LIN {X 0,Y 523.96,Z 519.214,A -85,B 0,C 180,E1 -4880.41,E2 -4880.41} C_VEL
LIN {X 0,Y 523.905,Z 519.224,A -85,B 0,C 180,E1 -4882.893,E2 -4882.893} C_VEL
LIN {X 0,Y 523.943,Z 519.224,A -85,B 0,C 180,E1 -4885.419,E2 -4885.419} C_VEL
LIN {X 0,Y 523.959,Z 519.22,A -85,B 0,C 180,E1 -4887.999,E2 -4887.999} C_VEL
LIN {X 0,Y 523.998,Z 519.419,A -85,B 0,C 180,E1 -4889.406,E2 -4889.406} C_VEL
LIN {X 0,Y 524.764,Z 524.163,A -85,B 0,C 180,E1 -4890.369,E2 -4890.369} C_VEL
LIN {X 0,Y 524.382,Z 539.428,A -85,B 0,C 180,E1 -4893.332,E2 -4893.332} C_VEL
LIN {X 0,Y 524.173,Z 547.59,A -85,B 0,C 180,E1 -4894.895,E2 -4894.895} C_VEL
LIN {X 0,Y 525.927,Z 557.88,A -85,B 0,C 180,E1 -4895.101,E2 -4895.101} C_VEL
LIN {X 0,Y 525.587,Z 637.04,A -85,B 0,C 180,E1 -4896.188,E2 -4896.188} C_VEL
LIN {X 0,Y 524.906,Z 640.968,A -85,B 0,C 180,E1 -4896.222,E2 -4896.222} C_VEL
LIN {X 0,Y 519.182,Z 653.237,A -85,B 0,C 180,E1 -4896.254,E2 -4896.254} C_VEL
LIN {X 0,Y 518.575,Z 657.117,A -85,B 0,C 180,E1 -4896.319,E2 -4896.319} C_VEL
LIN {X 0,Y 518.341,Z 670.235,A -85,B 0,C 180,E1 -4896.688,E2 -4896.688} C_VEL
LIN {X 0,Y 518.086,Z 682.787,A -85,B 0,C 180,E1 -4897.211,E2 -4897.211} C_VEL
LIN {X 0,Y 517.827,Z 694.371,A -85,B 0,C 180,E1 -4897.855,E2 -4897.855} C_VEL
LIN {X 0,Y 517.513,Z 705.687,A -85,B 0,C 180,E1 -4898.659,E2 -4898.659} C_VEL
LIN {X 0,Y 517.226,Z 715.845,A -85,B 0,C 180,E1 -4899.565,E2 -4899.565} C_VEL
LIN {X 0,Y 516.953,Z 724.842,A -85,B 0,C 180,E1 -4900.548,E2 -4900.548} C_VEL
LIN {X 0,Y 516.741,Z 732.6,A -85,B 0,C 180,E1 -4901.582,E2 -4901.582} C_VEL
LIN {X 0,Y 516.508,Z 740.372,A -85,B 0,C 180,E1 -4902.869,E2 -4902.869} C_VEL
LIN {X 0,Y 516.368,Z 746.561,A -85,B 0,C 180,E1 -4904.175,E2 -4904.175} C_VEL
LIN {X 0,Y 516.289,Z 751.444,A -85,B 0,C 180,E1 -4905.541,E2 -4905.541} C_VEL
LIN {X 0,Y 516.239,Z 754.36,A -85,B 0,C 180,E1 -4906.641,E2 -4906.641} C_VEL
LIN {X 0,Y 516.182,Z 756.998,A -85,B 0,C 180,E1 -4908.154,E2 -4908.154} C_VEL
LIN {X 0,Y 516.14,Z 758.095,A -85,B 0,C 180,E1 -4909.686,E2 -4909.686} C_VEL
LIN {X 0,Y 516.129,Z 757.71,A -85,B 0,C 180,E1 -4911.219,E2 -4911.219} C_VEL
LIN {X 0,Y 516.154,Z 756.609,A -85,B 0,C 180,E1 -4912.215,E2 -4912.215} C_VEL
LIN {X 0,Y 516.236,Z 754.376,A -85,B 0,C 180,E1 -4913.438,E2 -4913.438} C_VEL
LIN {X 0,Y 516.246,Z 750.774,A -85,B 0,C 180,E1 -4914.767,E2 -4914.767} C_VEL
LIN {X 0,Y 516.383,Z 745.673,A -85,B 0,C 180,E1 -4916.12,E2 -4916.12} C_VEL
LIN {X 0,Y 516.563,Z 738.759,A -85,B 0,C 180,E1 -4917.514,E2 -4917.514} C_VEL
LIN {X 0,Y 516.756,Z 731.562,A -85,B 0,C 180,E1 -4918.655,E2 -4918.655} C_VEL
LIN {X 0,Y 516.994,Z 722.592,A -85,B 0,C 180,E1 -4919.804,E2 -4919.804} C_VEL
LIN {X 0,Y 517.265,Z 712.654,A -85,B 0,C 180,E1 -4920.83,E2 -4920.83} C_VEL
LIN {X 0,Y 517.605,Z 701.844,A -85,B 0,C 180,E1 -4921.723,E2 -4921.723} C_VEL
LIN {X 0,Y 517.9,Z 691.117,A -85,B 0,C 180,E1 -4922.434,E2 -4922.434} C_VEL
LIN {X 0,Y 518.189,Z 679.448,A -85,B 0,C 180,E1 -4923.033,E2 -4923.033} C_VEL
LIN {X 0,Y 518.403,Z 666.182,A -85,B 0,C 180,E1 -4923.534,E2 -4923.534} C_VEL
LIN {X 0,Y 518.597,Z 653.698,A -85,B 0,C 180,E1 -4923.843,E2 -4923.843} C_VEL
LIN {X 0,Y 519.061,Z 558.357,A -85,B 0,C 180,E1 -4925.184,E2 -4925.184} C_VEL
LIN {X 0,Y 517.217,Z 547.636,A -85,B 0,C 180,E1 -4925.419,E2 -4925.419} C_VEL
LIN {X 0,Y 517.535,Z 532.885,A -85,B 0,C 180,E1 -4928.283,E2 -4928.283} C_VEL
LIN {X 0,Y 517.722,Z 524.988,A -85,B 0,C 180,E1 -4929.828,E2 -4929.828} C_VEL
LIN {X 0,Y 516.919,Z 520.098,A -85,B 0,C 180,E1 -4930.854,E2 -4930.854} C_VEL
LIN {X 0,Y 516.911,Z 520.095,A -85,B 0,C 180,E1 -4933.411,E2 -4933.411} C_VEL
LIN {X 0,Y 516.891,Z 520.095,A -85,B 0,C 180,E1 -4935.835,E2 -4935.835} C_VEL
LIN {X 0,Y 516.96,Z 520.086,A -85,B 0,C 180,E1 -4938.235,E2 -4938.235} C_VEL
LIN {X 0,Y 516.965,Z 520.086,A -85,B 0,C 180,E1 -4941.401,E2 -4941.401} C_VEL
LIN {X 0,Y 516.999,Z 520.08,A -85,B 0,C 180,E1 -4943.758,E2 -4943.758} C_VEL
LIN {X 0,Y 517.012,Z 520.088,A -85,B 0,C 180,E1 -4946.884,E2 -4946.884} C_VEL
LIN {X 0,Y 517.083,Z 520.069,A -85,B 0,C 180,E1 -4950.001,E2 -4950.001} C_VEL
LIN {X 0,Y 517.011,Z 520.085,A -85,B 0,C 180,E1 -4953.118,E2 -4953.118} C_VEL
LIN {X 0,Y 517,Z 520.08,A -85,B 0,C 180,E1 -4956.244,E2 -4956.244} C_VEL
LIN {X 0,Y 516.95,Z 520.09,A -85,B 0,C 180,E1 -4959.39,E2 -4959.39} C_VEL
LIN {X 0,Y 516.951,Z 520.086,A -85,B 0,C 180,E1 -4961.809,E2 -4961.809} C_VEL
LIN {X 0,Y 516.944,Z 520.095,A -85,B 0,C 180,E1 -4965.148,E2 -4965.148} C_VEL
LIN {X 0,Y 516.916,Z 520.09,A -85,B 0,C 180,E1 -4968.224,E2 -4968.224} C_VEL
LIN {X 0,Y 516.913,Z 520.094,A -85,B 0,C 180,E1 -4970.702,E2 -4970.702} C_VEL
LIN {X 0,Y 516.891,Z 520.093,A -85,B 0,C 180,E1 -4974.074,E2 -4974.074} C_VEL
LIN {X 0,Y 516.925,Z 520.091,A -85,B 0,C 180,E1 -4976.659,E2 -4976.659} C_VEL
LIN {X 0,Y 516.912,Z 520.095,A -85,B 0,C 180,E1 -4979.525,E2 -4979.525} C_VEL
LIN {X 0,Y 516.897,Z 520.093,A -85,B 0,C 180,E1 -4982.544,E2 -4982.544} C_VEL
LIN {X 0,Y 516.867,Z 520.105,A -85,B 0,C 180,E1 -4985.331,E2 -4985.331} C_VEL
LIN {X 0,Y 516.883,Z 520.095,A -85,B 0,C 180,E1 -4987.944,E2 -4987.944} C_VEL
LIN {X 0,Y 516.888,Z 520.095,A -85,B 0,C 180,E1 -4990.742,E2 -4990.742} C_VEL
LIN {X 0,Y 516.908,Z 520.093,A -85,B 0,C 180,E1 -4992.83,E2 -4992.83} C_VEL
LIN {X 0,Y 516.925,Z 520.093,A -85,B 0,C 180,E1 -4995.011,E2 -4995.011} C_VEL
LIN {X 0,Y 516.918,Z 520.09,A -85,B 0,C 180,E1 -4998.399,E2 -4998.399} C_VEL
LIN {X 0,Y 516.885,Z 520.101,A -85,B 0,C 180,E1 -5001.285,E2 -5001.285} C_VEL
LIN {X 0,Y 516.875,Z 520.096,A -85,B 0,C 180,E1 -5004.221,E2 -5004.221} C_VEL
LIN {X 0,Y 516.9,Z 520.095,A -85,B 0,C 180,E1 -5007.054,E2 -5007.054} C_VEL
LIN {X 0,Y 516.896,Z 520.098,A -85,B 0,C 180,E1 -5009.797,E2 -5009.797} C_VEL
LIN {X 0,Y 516.93,Z 520.088,A -85,B 0,C 180,E1 -5012.468,E2 -5012.468} C_VEL
LIN {X 0,Y 516.913,Z 520.093,A -85,B 0,C 180,E1 -5015.073,E2 -5015.073} C_VEL
LIN {X 0,Y 516.89,Z 520.093,A -85,B 0,C 180,E1 -5018.463,E2 -5018.463} C_VEL
LIN {X 0,Y 516.905,Z 520.092,A -85,B 0,C 180,E1 -5020.955,E2 -5020.955} C_VEL
LIN {X 0,Y 516.914,Z 520.096,A -85,B 0,C 180,E1 -5023.411,E2 -5023.411} C_VEL
LIN {X 0,Y 516.901,Z 520.099,A -85,B 0,C 180,E1 -5025.834,E2 -5025.834} C_VEL
LIN {X 0,Y 516.972,Z 520.085,A -85,B 0,C 180,E1 -5028.234,E2 -5028.234} C_VEL
LIN {X 0,Y 516.971,Z 520.087,A -85,B 0,C 180,E1 -5031.4,E2 -5031.4} C_VEL
LIN {X 0,Y 517.016,Z 520.087,A -85,B 0,C 180,E1 -5033.757,E2 -5033.757} C_VEL
LIN {X 0,Y 517.089,Z 520.076,A -85,B 0,C 180,E1 -5037.664,E2 -5037.664} C_VEL
LIN {X 0,Y 517.1,Z 520.067,A -85,B 0,C 180,E1 -5040.779,E2 -5040.779} C_VEL
LIN {X 0,Y 517.018,Z 520.078,A -85,B 0,C 180,E1 -5043.117,E2 -5043.117} C_VEL
LIN {X 0,Y 517.017,Z 520.082,A -85,B 0,C 180,E1 -5046.243,E2 -5046.243} C_VEL
LIN {X 0,Y 516.951,Z 520.088,A -85,B 0,C 180,E1 -5049.39,E2 -5049.39} C_VEL
LIN {X 0,Y 516.96,Z 520.092,A -85,B 0,C 180,E1 -5051.807,E2 -5051.807} C_VEL
LIN {X 0,Y 516.952,Z 520.086,A -85,B 0,C 180,E1 -5055.147,E2 -5055.147} C_VEL
LIN {X 0,Y 516.924,Z 520.095,A -85,B 0,C 180,E1 -5058.223,E2 -5058.223} C_VEL
LIN {X 0,Y 516.92,Z 520.091,A -85,B 0,C 180,E1 -5060.702,E2 -5060.702} C_VEL
LIN {X 0,Y 516.898,Z 520.102,A -85,B 0,C 180,E1 -5064.073,E2 -5064.073} C_VEL
LIN {X 0,Y 516.93,Z 520.09,A -85,B 0,C 180,E1 -5066.658,E2 -5066.658} C_VEL
LIN {X 0,Y 516.919,Z 520.091,A -85,B 0,C 180,E1 -5069.524,E2 -5069.524} C_VEL
LIN {X 0,Y 516.901,Z 520.096,A -85,B 0,C 180,E1 -5072.543,E2 -5072.543} C_VEL
LIN {X 0,Y 516.884,Z 520.094,A -85,B 0,C 180,E1 -5075.331,E2 -5075.331} C_VEL
LIN {X 0,Y 516.888,Z 520.099,A -85,B 0,C 180,E1 -5077.943,E2 -5077.943} C_VEL
LIN {X 0,Y 516.889,Z 520.096,A -85,B 0,C 180,E1 -5080.742,E2 -5080.742} C_VEL
LIN {X 0,Y 516.888,Z 520.097,A -85,B 0,C 180,E1 -5083.903,E2 -5083.903} C_VEL
LIN {X 0,Y 516.889,Z 520.1,A -85,B 0,C 180,E1 -5086.107,E2 -5086.107} C_VEL
LIN {X 0,Y 516.921,Z 520.098,A -85,B 0,C 180,E1 -5088.398,E2 -5088.398} C_VEL
LIN {X 0,Y 516.887,Z 520.094,A -85,B 0,C 180,E1 -5091.284,E2 -5091.284} C_VEL
LIN {X 0,Y 516.878,Z 520.102,A -85,B 0,C 180,E1 -5094.219,E2 -5094.219} C_VEL
LIN {X 0,Y 516.902,Z 520.093,A -85,B 0,C 180,E1 -5097.052,E2 -5097.052} C_VEL
LIN {X 0,Y 516.899,Z 520.095,A -85,B 0,C 180,E1 -5099.796,E2 -5099.796} C_VEL
LIN {X 0,Y 516.934,Z 520.096,A -85,B 0,C 180,E1 -5102.467,E2 -5102.467} C_VEL
LIN {X 0,Y 516.925,Z 520.096,A -85,B 0,C 180,E1 -5105.397,E2 -5105.397} C_VEL
LIN {X 0,Y 516.918,Z 520.182,A -85,B 0,C 180,E1 -5105.595,E2 -5105.595} C_VEL
LIN {X 0,Y 518.517,Z 529.143,A -85,B 0,C 180,E1 -5107.173,E2 -5107.173} C_VEL
LIN {X 0,Y 518.016,Z 547.542,A -85,B 0,C 180,E1 -5110.172,E2 -5110.172} C_VEL
LIN {X 0,Y 517.581,Z 564.071,A -85,B 0,C 180,E1 -5112.821,E2 -5112.821} C_VEL
LIN {X 0,Y 517.335,Z 575.468,A -85,B 0,C 180,E1 -5114.64,E2 -5114.64} C_VEL
LIN {X 0,Y 519.112,Z 587.664,A -85,B 0,C 180,E1 -5114.867,E2 -5114.867} C_VEL
LIN {X 0,Y 518.603,Z 684.232,A -85,B 0,C 180,E1 -5116.23,E2 -5116.23} C_VEL
LIN {X 0,Y 518.342,Z 698.045,A -85,B 0,C 180,E1 -5116.598,E2 -5116.598} C_VEL
LIN {X 0,Y 518.105,Z 710.943,A -85,B 0,C 180,E1 -5117.115,E2 -5117.115} C_VEL
LIN {X 0,Y 517.775,Z 722.904,A -85,B 0,C 180,E1 -5117.767,E2 -5117.767} C_VEL
LIN {X 0,Y 517.531,Z 734.057,A -85,B 0,C 180,E1 -5118.544,E2 -5118.544} C_VEL
LIN {X 0,Y 517.18,Z 744.285,A -85,B 0,C 180,E1 -5119.428,E2 -5119.428} C_VEL
LIN {X 0,Y 516.953,Z 753.482,A -85,B 0,C 180,E1 -5120.412,E2 -5120.412} C_VEL
LIN {X 0,Y 516.686,Z 762.438,A -85,B 0,C 180,E1 -5121.591,E2 -5121.591} C_VEL
LIN {X 0,Y 516.512,Z 769.646,A -85,B 0,C 180,E1 -5122.768,E2 -5122.768} C_VEL
LIN {X 0,Y 516.455,Z 776.211,A -85,B 0,C 180,E1 -5124.141,E2 -5124.141} C_VEL
LIN {X 0,Y 516.272,Z 780.548,A -85,B 0,C 180,E1 -5125.314,E2 -5125.314} C_VEL
LIN {X 0,Y 516.355,Z 782.848,A -85,B 0,C 180,E1 -5126.097,E2 -5126.097} C_VEL
LIN {X 0,Y 516.283,Z 784.709,A -85,B 0,C 180,E1 -5126.878,E2 -5126.878} C_VEL
LIN {X 0,Y 516.261,Z 786.105,A -85,B 0,C 180,E1 -5127.658,E2 -5127.658} C_VEL
LIN {X 0,Y 516.16,Z 787.707,A -85,B 0,C 180,E1 -5129.219,E2 -5129.219} C_VEL
LIN {X 0,Y 516.154,Z 787.924,A -85,B 0,C 180,E1 -5129.999,E2 -5129.999} C_VEL
LIN {X 0,Y 516.192,Z 787.103,A -85,B 0,C 180,E1 -5131.559,E2 -5131.559} C_VEL
LIN {X 0,Y 516.26,Z 786.11,A -85,B 0,C 180,E1 -5132.339,E2 -5132.339} C_VEL
LIN {X 0,Y 516.282,Z 784.715,A -85,B 0,C 180,E1 -5133.12,E2 -5133.12} C_VEL
LIN {X 0,Y 516.326,Z 781.78,A -85,B 0,C 180,E1 -5134.292,E2 -5134.292} C_VEL
LIN {X 0,Y 516.405,Z 777.806,A -85,B 0,C 180,E1 -5135.465,E2 -5135.465} C_VEL
LIN {X 0,Y 516.462,Z 772.519,A -85,B 0,C 180,E1 -5136.676,E2 -5136.676} C_VEL
LIN {X 0,Y 516.596,Z 766.242,A -85,B 0,C 180,E1 -5137.818,E2 -5137.818} C_VEL
LIN {X 0,Y 516.809,Z 758.201,A -85,B 0,C 180,E1 -5138.996,E2 -5138.996} C_VEL
LIN {X 0,Y 517.023,Z 750.003,A -85,B 0,C 180,E1 -5139.979,E2 -5139.979} C_VEL
LIN {X 0,Y 517.326,Z 740.004,A -85,B 0,C 180,E1 -5140.963,E2 -5140.963} C_VEL
LIN {X 0,Y 517.655,Z 728.793,A -85,B 0,C 180,E1 -5141.842,E2 -5141.842} C_VEL
LIN {X 0,Y 517.961,Z 717.633,A -85,B 0,C 180,E1 -5142.537,E2 -5142.537} C_VEL
LIN {X 0,Y 518.237,Z 705.353,A -85,B 0,C 180,E1 -5143.128,E2 -5143.128} C_VEL
LIN {X 0,Y 518.456,Z 692.405,A -85,B 0,C 180,E1 -5143.572,E2 -5143.572} C_VEL
LIN {X 0,Y 518.687,Z 678.625,A -85,B 0,C 180,E1 -5143.865,E2 -5143.865} C_VEL
LIN {X 0,Y 518.996,Z 585.709,A -85,B 0,C 180,E1 -5145.163,E2 -5145.163} C_VEL
LIN {X 0,Y 517.345,Z 575.322,A -85,B 0,C 180,E1 -5145.367,E2 -5145.367} C_VEL
LIN {X 0,Y 517.811,Z 555.065,A -85,B 0,C 180,E1 -5148.598,E2 -5148.598} C_VEL
LIN {X 0,Y 518.244,Z 537.216,A -85,B 0,C 180,E1 -5151.477,E2 -5151.477} C_VEL
LIN {X 0,Y 518.501,Z 528.987,A -85,B 0,C 180,E1 -5152.823,E2 -5152.823} C_VEL
LIN {X 0,Y 516.92,Z 520.096,A -85,B 0,C 180,E1 -5154.406,E2 -5154.406} C_VEL
LIN {X 0,Y 516.925,Z 520.093,A -85,B 0,C 180,E1 -5156.656,E2 -5156.656} C_VEL
LIN {X 0,Y 516.909,Z 520.102,A -85,B 0,C 180,E1 -5159.523,E2 -5159.523} C_VEL
LIN {X 0,Y 516.898,Z 520.095,A -85,B 0,C 180,E1 -5162.543,E2 -5162.543} C_VEL
LIN {X 0,Y 516.876,Z 520.104,A -85,B 0,C 180,E1 -5165.331,E2 -5165.331} C_VEL
LIN {X 0,Y 516.878,Z 520.1,A -85,B 0,C 180,E1 -5167.942,E2 -5167.942} C_VEL
LIN {X 0,Y 516.881,Z 520.098,A -85,B 0,C 180,E1 -5170.74,E2 -5170.74} C_VEL
LIN {X 0,Y 516.899,Z 520.096,A -85,B 0,C 180,E1 -5172.828,E2 -5172.828} C_VEL
LIN {X 0,Y 516.916,Z 520.095,A -85,B 0,C 180,E1 -5175.009,E2 -5175.009} C_VEL
LIN {X 0,Y 516.916,Z 520.092,A -85,B 0,C 180,E1 -5178.396,E2 -5178.396} C_VEL
LIN {X 0,Y 516.88,Z 520.102,A -85,B 0,C 180,E1 -5181.284,E2 -5181.284} C_VEL
LIN {X 0,Y 516.885,Z 520.095,A -85,B 0,C 180,E1 -5184.22,E2 -5184.22} C_VEL
LIN {X 0,Y 516.89,Z 520.097,A -85,B 0,C 180,E1 -5187.052,E2 -5187.052} C_VEL
LIN {X 0,Y 516.894,Z 520.098,A -85,B 0,C 180,E1 -5189.796,E2 -5189.796} C_VEL
LIN {X 0,Y 516.921,Z 520.089,A -85,B 0,C 180,E1 -5192.467,E2 -5192.467} C_VEL
LIN {X 0,Y 516.903,Z 520.097,A -85,B 0,C 180,E1 -5195.071,E2 -5195.071} C_VEL
LIN {X 0,Y 516.877,Z 520.096,A -85,B 0,C 180,E1 -5198.461,E2 -5198.461} C_VEL
LIN {X 0,Y 516.895,Z 520.093,A -85,B 0,C 180,E1 -5200.954,E2 -5200.954} C_VEL
LIN {X 0,Y 516.908,Z 520.099,A -85,B 0,C 180,E1 -5203.41,E2 -5203.41} C_VEL
LIN {X 0,Y 516.896,Z 520.097,A -85,B 0,C 180,E1 -5205.833,E2 -5205.833} C_VEL
LIN {X 0,Y 516.993,Z 520.08,A -85,B 0,C 180,E1 -5208.234,E2 -5208.234} C_VEL
LIN {X 0,Y 516.962,Z 520.092,A -85,B 0,C 180,E1 -5211.399,E2 -5211.399} C_VEL
LIN {X 0,Y 517,Z 520.084,A -85,B 0,C 180,E1 -5213.756,E2 -5213.756} C_VEL
LIN {X 0,Y 517.007,Z 520.081,A -85,B 0,C 180,E1 -5216.883,E2 -5216.883} C_VEL
LIN {X 0,Y 517.074,Z 520.073,A -85,B 0,C 180,E1 -5220,E2 -5220} C_VEL
LIN {X 0,Y 517.007,Z 520.084,A -85,B 0,C 180,E1 -5223.117,E2 -5223.117} C_VEL
LIN {X 0,Y 516.999,Z 520.081,A -85,B 0,C 180,E1 -5226.243,E2 -5226.243} C_VEL
LIN {X 0,Y 516.947,Z 520.095,A -85,B 0,C 180,E1 -5229.389,E2 -5229.389} C_VEL
LIN {X 0,Y 516.971,Z 520.088,A -85,B 0,C 180,E1 -5231.824,E2 -5231.824} C_VEL
LIN {X 0,Y 516.931,Z 520.096,A -85,B 0,C 180,E1 -5235.146,E2 -5235.146} C_VEL
LIN {X 0,Y 516.914,Z 520.093,A -85,B 0,C 180,E1 -5238.222,E2 -5238.222} C_VEL
LIN {X 0,Y 516.901,Z 520.095,A -85,B 0,C 180,E1 -5240.701,E2 -5240.701} C_VEL
LIN {X 0,Y 516.899,Z 520.096,A -85,B 0,C 180,E1 -5244.072,E2 -5244.072} C_VEL
LIN {X 0,Y 516.917,Z 520.094,A -85,B 0,C 180,E1 -5246.658,E2 -5246.658} C_VEL
LIN {X 0,Y 516.949,Z 520.261,A -85,B 0,C 180,E1 -5249.246,E2 -5249.246} C_VEL
LIN {X 0,Y 517.804,Z 525.726,A -85,B 0,C 180,E1 -5250.37,E2 -5250.37} C_VEL
LIN {X 0,Y 517.38,Z 541.055,A -85,B 0,C 180,E1 -5253.376,E2 -5253.376} C_VEL
LIN {X 0,Y 517.2,Z 547.848,A -85,B 0,C 180,E1 -5254.694,E2 -5254.694} C_VEL
LIN {X 0,Y 519.105,Z 559.366,A -85,B 0,C 180,E1 -5254.919,E2 -5254.919} C_VEL
LIN {X 0,Y 518.611,Z 654.9,A -85,B 0,C 180,E1 -5256.271,E2 -5256.271} C_VEL
LIN {X 0,Y 518.575,Z 657.117,A -85,B 0,C 180,E1 -5256.319,E2 -5256.319} C_VEL
LIN {X 0,Y 517.98,Z 662.864,A -85,B 0,C 180,E1 -5256.446,E2 -5256.446} C_VEL
LIN {X 0,Y 515.1,Z 672.116,A -85,B 0,C 180,E1 -5256.671,E2 -5256.671} C_VEL
LIN {X 0,Y 511.993,Z 681.148,A -85,B 0,C 180,E1 -5256.969,E2 -5256.969} C_VEL
LIN {X 0,Y 511.092,Z 686.554,A -85,B 0,C 180,E1 -5257.22,E2 -5257.22} C_VEL
LIN {X 0,Y 510.843,Z 697.349,A -85,B 0,C 180,E1 -5257.874,E2 -5257.874} C_VEL
LIN {X 0,Y 510.482,Z 707.734,A -85,B 0,C 180,E1 -5258.659,E2 -5258.659} C_VEL
LIN {X 0,Y 510.18,Z 718.534,A -85,B 0,C 180,E1 -5259.678,E2 -5259.678} C_VEL
LIN {X 0,Y 509.819,Z 728.328,A -85,B 0,C 180,E1 -5260.838,E2 -5260.838} C_VEL
LIN {X 0,Y 509.594,Z 735.386,A -85,B 0,C 180,E1 -5261.866,E2 -5261.866} C_VEL
LIN {X 0,Y 509.404,Z 741.838,A -85,B 0,C 180,E1 -5263.014,E2 -5263.014} C_VEL
LIN {X 0,Y 509.296,Z 748.002,A -85,B 0,C 180,E1 -5264.411,E2 -5264.411} C_VEL
LIN {X 0,Y 509.186,Z 752.773,A -85,B 0,C 180,E1 -5265.866,E2 -5265.866} C_VEL
LIN {X 0,Y 509.095,Z 756.203,A -85,B 0,C 180,E1 -5267.436,E2 -5267.436} C_VEL
LIN {X 0,Y 509.069,Z 757.591,A -85,B 0,C 180,E1 -5268.498,E2 -5268.498} C_VEL
LIN {X 0,Y 509.057,Z 758.272,A -85,B 0,C 180,E1 -5269.545,E2 -5269.545} C_VEL
LIN {X 0,Y 509.057,Z 758.251,A -85,B 0,C 180,E1 -5270.635,E2 -5270.635} C_VEL
LIN {X 0,Y 509.064,Z 757.277,A -85,B 0,C 180,E1 -5271.898,E2 -5271.898} C_VEL
LIN {X 0,Y 509.114,Z 755.211,A -85,B 0,C 180,E1 -5273.192,E2 -5273.192} C_VEL
LIN {X 0,Y 509.183,Z 751.755,A -85,B 0,C 180,E1 -5274.572,E2 -5274.572} C_VEL
LIN {X 0,Y 509.29,Z 747.169,A -85,B 0,C 180,E1 -5275.89,E2 -5275.89} C_VEL
LIN {X 0,Y 509.455,Z 740.661,A -85,B 0,C 180,E1 -5277.298,E2 -5277.298} C_VEL
LIN {X 0,Y 509.673,Z 732.901,A -85,B 0,C 180,E1 -5278.605,E2 -5278.605} C_VEL
LIN {X 0,Y 509.945,Z 723.931,A -85,B 0,C 180,E1 -5279.801,E2 -5279.801} C_VEL
LIN {X 0,Y 510.235,Z 714.274,A -85,B 0,C 180,E1 -5280.841,E2 -5280.841} C_VEL
LIN {X 0,Y 510.563,Z 703.645,A -85,B 0,C 180,E1 -5281.759,E2 -5281.759} C_VEL
LIN {X 0,Y 510.95,Z 691.902,A -85,B 0,C 180,E1 -5282.564,E2 -5282.564} C_VEL
LIN {X 0,Y 511.282,Z 679.617,A -85,B 0,C 180,E1 -5283.208,E2 -5283.208} C_VEL
LIN {X 0,Y 511.512,Z 666.516,A -85,B 0,C 180,E1 -5283.71,E2 -5283.71} C_VEL
LIN {X 0,Y 511.725,Z 653.986,A -85,B 0,C 180,E1 -5284.026,E2 -5284.026} C_VEL
LIN {X 0,Y 512.146,Z 558.762,A -85,B 0,C 180,E1 -5285.389,E2 -5285.389} C_VEL
LIN {X 0,Y 510.224,Z 547.903,A -85,B 0,C 180,E1 -5285.621,E2 -5285.621} C_VEL
LIN {X 0,Y 510.56,Z 533.785,A -85,B 0,C 180,E1 -5288.395,E2 -5288.395} C_VEL
LIN {X 0,Y 510.76,Z 526.274,A -85,B 0,C 180,E1 -5289.881,E2 -5289.881} C_VEL
LIN {X 0,Y 509.865,Z 520.976,A -85,B 0,C 180,E1 -5290.997,E2 -5290.997} C_VEL
LIN {X 0,Y 509.879,Z 520.973,A -85,B 0,C 180,E1 -5293.176,E2 -5293.176} C_VEL
LIN {X 0,Y 509.859,Z 520.971,A -85,B 0,C 180,E1 -5295.635,E2 -5295.635} C_VEL
LIN {X 0,Y 509.897,Z 520.965,A -85,B 0,C 180,E1 -5298.124,E2 -5298.124} C_VEL
LIN {X 0,Y 509.912,Z 520.966,A -85,B 0,C 180,E1 -5301.281,E2 -5301.281} C_VEL
LIN {X 0,Y 509.95,Z 520.958,A -85,B 0,C 180,E1 -5303.671,E2 -5303.671} C_VEL
LIN {X 0,Y 509.954,Z 520.966,A -85,B 0,C 180,E1 -5306.841,E2 -5306.841} C_VEL
LIN {X 0,Y 510.061,Z 520.949,A -85,B 0,C 180,E1 -5309.212,E2 -5309.212} C_VEL
LIN {X 0,Y 510.054,Z 520.947,A -85,B 0,C 180,E1 -5312.37,E2 -5312.37} C_VEL
LIN {X 0,Y 509.977,Z 520.956,A -85,B 0,C 180,E1 -5315.537,E2 -5315.537} C_VEL
LIN {X 0,Y 509.95,Z 520.958,A -85,B 0,C 180,E1 -5317.923,E2 -5317.923} C_VEL
LIN {X 0,Y 509.912,Z 520.971,A -85,B 0,C 180,E1 -5321.127,E2 -5321.127} C_VEL
LIN {X 0,Y 509.868,Z 520.971,A -85,B 0,C 180,E1 -5323.553,E2 -5323.553} C_VEL
LIN {X 0,Y 509.852,Z 520.97,A -85,B 0,C 180,E1 -5326.004,E2 -5326.004} C_VEL
LIN {X 0,Y 509.862,Z 520.97,A -85,B 0,C 180,E1 -5328.485,E2 -5328.485} C_VEL
LIN {X 0,Y 509.85,Z 520.978,A -85,B 0,C 180,E1 -5331.003,E2 -5331.003} C_VEL
LIN {X 0,Y 509.855,Z 520.97,A -85,B 0,C 180,E1 -5334.428,E2 -5334.428} C_VEL
LIN {X 0,Y 509.884,Z 520.973,A -85,B 0,C 180,E1 -5337.057,E2 -5337.057} C_VEL
LIN {X 0,Y 509.858,Z 520.971,A -85,B 0,C 180,E1 -5339.752,E2 -5339.752} C_VEL
LIN {X 0,Y 509.874,Z 520.97,A -85,B 0,C 180,E1 -5342.775,E2 -5342.775} C_VEL
LIN {X 0,Y 509.827,Z 520.978,A -85,B 0,C 180,E1 -5345.579,E2 -5345.579} C_VEL
LIN {X 0,Y 509.852,Z 520.97,A -85,B 0,C 180,E1 -5348.339,E2 -5348.339} C_VEL
LIN {X 0,Y 509.861,Z 520.977,A -85,B 0,C 180,E1 -5351.426,E2 -5351.426} C_VEL
LIN {X 0,Y 509.86,Z 520.97,A -85,B 0,C 180,E1 -5354.669,E2 -5354.669} C_VEL
LIN {X 0,Y 509.859,Z 520.97,A -85,B 0,C 180,E1 -5358.104,E2 -5358.104} C_VEL
LIN {X 0,Y 509.85,Z 520.971,A -85,B 0,C 180,E1 -5360.649,E2 -5360.649} C_VEL
LIN {X 0,Y 509.828,Z 520.979,A -85,B 0,C 180,E1 -5363.648,E2 -5363.648} C_VEL
LIN {X 0,Y 509.864,Z 520.969,A -85,B 0,C 180,E1 -5366.54,E2 -5366.54} C_VEL
LIN {X 0,Y 509.849,Z 520.977,A -85,B 0,C 180,E1 -5369.335,E2 -5369.335} C_VEL
LIN {X 0,Y 509.896,Z 520.967,A -85,B 0,C 180,E1 -5372.055,E2 -5372.055} C_VEL
LIN {X 0,Y 509.881,Z 520.967,A -85,B 0,C 180,E1 -5374.705,E2 -5374.705} C_VEL
LIN {X 0,Y 509.832,Z 520.98,A -85,B 0,C 180,E1 -5377.459,E2 -5377.459} C_VEL
LIN {X 0,Y 509.922,Z 520.967,A -85,B 0,C 180,E1 -5379.845,E2 -5379.845} C_VEL
LIN {X 0,Y 509.881,Z 520.969,A -85,B 0,C 180,E1 -5383.175,E2 -5383.175} C_VEL
LIN {X 0,Y 509.87,Z 520.977,A -85,B 0,C 180,E1 -5385.635,E2 -5385.635} C_VEL
LIN {X 0,Y 509.919,Z 520.962,A -85,B 0,C 180,E1 -5388.875,E2 -5388.875} C_VEL
LIN {X 0,Y 509.957,Z 520.961,A -85,B 0,C 180,E1 -5392.079,E2 -5392.079} C_VEL
LIN {X 0,Y 509.987,Z 520.954,A -85,B 0,C 180,E1 -5394.465,E2 -5394.465} C_VEL
LIN {X 0,Y 510.06,Z 520.951,A -85,B 0,C 180,E1 -5397.631,E2 -5397.631} C_VEL
LIN {X 0,Y 510.07,Z 520.943,A -85,B 0,C 180,E1 -5400.79,E2 -5400.79} C_VEL
LIN {X 0,Y 509.96,Z 520.957,A -85,B 0,C 180,E1 -5403.16,E2 -5403.16} C_VEL
LIN {X 0,Y 509.986,Z 520.956,A -85,B 0,C 180,E1 -5406.33,E2 -5406.33} C_VEL
LIN {X 0,Y 509.918,Z 520.962,A -85,B 0,C 180,E1 -5408.721,E2 -5408.721} C_VEL
LIN {X 0,Y 509.912,Z 520.972,A -85,B 0,C 180,E1 -5411.932,E2 -5411.932} C_VEL
LIN {X 0,Y 509.902,Z 520.964,A -85,B 0,C 180,E1 -5415.242,E2 -5415.242} C_VEL
LIN {X 0,Y 509.874,Z 520.977,A -85,B 0,C 180,E1 -5417.993,E2 -5417.993} C_VEL
LIN {X 0,Y 509.894,Z 520.969,A -85,B 0,C 180,E1 -5420.401,E2 -5420.401} C_VEL
LIN {X 0,Y 509.83,Z 520.975,A -85,B 0,C 180,E1 -5423.564,E2 -5423.564} C_VEL
LIN {X 0,Y 509.918,Z 520.967,A -85,B 0,C 180,E1 -5426.378,E2 -5426.378} C_VEL
LIN {X 0,Y 509.882,Z 520.967,A -85,B 0,C 180,E1 -5428.844,E2 -5428.844} C_VEL
LIN {X 0,Y 509.827,Z 520.975,A -85,B 0,C 180,E1 -5431.59,E2 -5431.59} C_VEL
LIN {X 0,Y 509.849,Z 520.976,A -85,B 0,C 180,E1 -5434.414,E2 -5434.414} C_VEL
LIN {X 0,Y 509.826,Z 520.973,A -85,B 0,C 180,E1 -5437.34,E2 -5437.34} C_VEL
LIN {X 0,Y 509.845,Z 520.978,A -85,B 0,C 180,E1 -5440.382,E2 -5440.382} C_VEL
LIN {X 0,Y 509.808,Z 520.976,A -85,B 0,C 180,E1 -5443.059,E2 -5443.059} C_VEL
LIN {X 0,Y 509.83,Z 520.975,A -85,B 0,C 180,E1 -5445.793,E2 -5445.793} C_VEL
LIN {X 0,Y 509.862,Z 520.974,A -85,B 0,C 180,E1 -5448.574,E2 -5448.574} C_VEL
LIN {X 0,Y 509.858,Z 520.971,A -85,B 0,C 180,E1 -5451.786,E2 -5451.786} C_VEL
LIN {X 0,Y 509.837,Z 520.977,A -85,B 0,C 180,E1 -5454.621,E2 -5454.621} C_VEL
LIN {X 0,Y 509.868,Z 520.968,A -85,B 0,C 180,E1 -5457.48,E2 -5457.48} C_VEL
LIN {X 0,Y 509.865,Z 520.977,A -85,B 0,C 180,E1 -5460.273,E2 -5460.273} C_VEL
LIN {X 0,Y 509.892,Z 520.97,A -85,B 0,C 180,E1 -5462.944,E2 -5462.944} C_VEL
LIN {X 0,Y 509.924,Z 521.127,A -85,B 0,C 180,E1 -5465.424,E2 -5465.424} C_VEL
LIN {X 0,Y 511.571,Z 530.707,A -85,B 0,C 180,E1 -5467.132,E2 -5467.132} C_VEL
LIN {X 0,Y 511.041,Z 548.651,A -85,B 0,C 180,E1 -5470.1,E2 -5470.1} C_VEL
LIN {X 0,Y 510.56,Z 565.156,A -85,B 0,C 180,E1 -5472.784,E2 -5472.784} C_VEL
LIN {X 0,Y 510.34,Z 575.214,A -85,B 0,C 180,E1 -5474.414,E2 -5474.414} C_VEL
LIN {X 0,Y 512.245,Z 587.917,A -85,B 0,C 180,E1 -5474.667,E2 -5474.667} C_VEL
LIN {X 0,Y 511.735,Z 683.859,A -85,B 0,C 180,E1 -5476.042,E2 -5476.042} C_VEL
LIN {X 0,Y 511.444,Z 696.962,A -85,B 0,C 180,E1 -5476.388,E2 -5476.388} C_VEL
LIN {X 0,Y 511.191,Z 709.611,A -85,B 0,C 180,E1 -5476.887,E2 -5476.887} C_VEL
LIN {X 0,Y 510.865,Z 721.069,A -85,B 0,C 180,E1 -5477.499,E2 -5477.499} C_VEL
LIN {X 0,Y 510.581,Z 732.509,A -85,B 0,C 180,E1 -5478.285,E2 -5478.285} C_VEL
LIN {X 0,Y 510.242,Z 742.993,A -85,B 0,C 180,E1 -5479.182,E2 -5479.182} C_VEL
LIN {X 0,Y 509.971,Z 751.563,A -85,B 0,C 180,E1 -5480.079,E2 -5480.079} C_VEL
LIN {X 0,Y 509.712,Z 759.467,A -85,B 0,C 180,E1 -5481.075,E2 -5481.075} C_VEL
LIN {X 0,Y 509.515,Z 767.187,A -85,B 0,C 180,E1 -5482.27,E2 -5482.27} C_VEL
LIN {X 0,Y 509.329,Z 774.295,A -85,B 0,C 180,E1 -5483.661,E2 -5483.661} C_VEL
LIN {X 0,Y 509.248,Z 779.025,A -85,B 0,C 180,E1 -5484.852,E2 -5484.852} C_VEL
LIN {X 0,Y 509.25,Z 782.64,A -85,B 0,C 180,E1 -5486.042,E2 -5486.042} C_VEL
LIN {X 0,Y 509.201,Z 784.504,A -85,B 0,C 180,E1 -5486.834,E2 -5486.834} C_VEL
LIN {X 0,Y 509.189,Z 785.901,A -85,B 0,C 180,E1 -5487.626,E2 -5487.626} C_VEL
LIN {X 0,Y 509.074,Z 787.503,A -85,B 0,C 180,E1 -5489.208,E2 -5489.208} C_VEL
LIN {X 0,Y 509.065,Z 787.719,A -85,B 0,C 180,E1 -5489.999,E2 -5489.999} C_VEL
LIN {X 0,Y 509.112,Z 786.897,A -85,B 0,C 180,E1 -5491.581,E2 -5491.581} C_VEL
LIN {X 0,Y 509.189,Z 785.903,A -85,B 0,C 180,E1 -5492.372,E2 -5492.372} C_VEL
LIN {X 0,Y 509.2,Z 784.504,A -85,B 0,C 180,E1 -5493.164,E2 -5493.164} C_VEL
LIN {X 0,Y 509.216,Z 781.564,A -85,B 0,C 180,E1 -5494.352,E2 -5494.352} C_VEL
LIN {X 0,Y 509.322,Z 777.586,A -85,B 0,C 180,E1 -5495.542,E2 -5495.542} C_VEL
LIN {X 0,Y 509.4,Z 771.917,A -85,B 0,C 180,E1 -5496.843,E2 -5496.843} C_VEL
LIN {X 0,Y 509.572,Z 764.77,A -85,B 0,C 180,E1 -5498.126,E2 -5498.126} C_VEL
LIN {X 0,Y 509.793,Z 756.462,A -85,B 0,C 180,E1 -5499.321,E2 -5499.321} C_VEL
LIN {X 0,Y 510.033,Z 747.941,A -85,B 0,C 180,E1 -5500.318,E2 -5500.318} C_VEL
LIN {X 0,Y 510.435,Z 737.415,A -85,B 0,C 180,E1 -5501.314,E2 -5501.314} C_VEL
LIN {X 0,Y 510.723,Z 726.404,A -85,B 0,C 180,E1 -5502.154,E2 -5502.154} C_VEL
LIN {X 0,Y 511.054,Z 715.558,A -85,B 0,C 180,E1 -5502.811,E2 -5502.811} C_VEL
LIN {X 0,Y 511.324,Z 703.775,A -85,B 0,C 180,E1 -5503.36,E2 -5503.36} C_VEL
LIN {X 0,Y 511.59,Z 690.19,A -85,B 0,C 180,E1 -5503.808,E2 -5503.808} C_VEL
LIN {X 0,Y 511.795,Z 676.51,A -85,B 0,C 180,E1 -5504.081,E2 -5504.081} C_VEL
LIN {X 0,Y 512.072,Z 586.153,A -85,B 0,C 180,E1 -5505.363,E2 -5505.363} C_VEL
LIN {X 0,Y 510.329,Z 575.072,A -85,B 0,C 180,E1 -5505.587,E2 -5505.587} C_VEL
LIN {X 0,Y 510.856,Z 554.834,A -85,B 0,C 180,E1 -5508.861,E2 -5508.861} C_VEL
LIN {X 0,Y 511.373,Z 535.755,A -85,B 0,C 180,E1 -5511.992,E2 -5511.992} C_VEL
LIN {X 0,Y 511.511,Z 529.767,A -85,B 0,C 180,E1 -5512.991,E2 -5512.991} C_VEL
LIN {X 0,Y 509.874,Z 520.975,A -85,B 0,C 180,E1 -5514.571,E2 -5514.571} C_VEL
LIN {X 0,Y 509.884,Z 520.973,A -85,B 0,C 180,E1 -5517.054,E2 -5517.054} C_VEL
LIN {X 0,Y 509.855,Z 520.979,A -85,B 0,C 180,E1 -5519.75,E2 -5519.75} C_VEL
LIN {X 0,Y 509.874,Z 520.971,A -85,B 0,C 180,E1 -5522.773,E2 -5522.773} C_VEL
LIN {X 0,Y 509.836,Z 520.981,A -85,B 0,C 180,E1 -5525.579,E2 -5525.579} C_VEL
LIN {X 0,Y 509.855,Z 520.972,A -85,B 0,C 180,E1 -5528.336,E2 -5528.336} C_VEL
LIN {X 0,Y 509.854,Z 520.981,A -85,B 0,C 180,E1 -5531.424,E2 -5531.424} C_VEL
LIN {X 0,Y 509.851,Z 520.973,A -85,B 0,C 180,E1 -5534.667,E2 -5534.667} C_VEL
LIN {X 0,Y 509.854,Z 520.973,A -85,B 0,C 180,E1 -5538.101,E2 -5538.101} C_VEL
LIN {X 0,Y 509.853,Z 520.971,A -85,B 0,C 180,E1 -5540.648,E2 -5540.648} C_VEL
LIN {X 0,Y 509.829,Z 520.98,A -85,B 0,C 180,E1 -5543.647,E2 -5543.647} C_VEL
LIN {X 0,Y 509.856,Z 520.97,A -85,B 0,C 180,E1 -5546.538,E2 -5546.538} C_VEL
LIN {X 0,Y 509.842,Z 520.978,A -85,B 0,C 180,E1 -5549.334,E2 -5549.334} C_VEL
LIN {X 0,Y 509.887,Z 520.966,A -85,B 0,C 180,E1 -5552.054,E2 -5552.054} C_VEL
LIN {X 0,Y 509.869,Z 520.97,A -85,B 0,C 180,E1 -5554.703,E2 -5554.703} C_VEL
LIN {X 0,Y 509.846,Z 520.978,A -85,B 0,C 180,E1 -5557.449,E2 -5557.449} C_VEL
LIN {X 0,Y 509.907,Z 520.964,A -85,B 0,C 180,E1 -5559.844,E2 -5559.844} C_VEL
LIN {X 0,Y 509.877,Z 520.973,A -85,B 0,C 180,E1 -5563.174,E2 -5563.174} C_VEL
LIN {X 0,Y 509.863,Z 520.976,A -85,B 0,C 180,E1 -5565.634,E2 -5565.634} C_VEL
LIN {X 0,Y 509.915,Z 520.963,A -85,B 0,C 180,E1 -5568.874,E2 -5568.874} C_VEL
LIN {X 0,Y 509.941,Z 520.96,A -85,B 0,C 180,E1 -5572.078,E2 -5572.078} C_VEL
LIN {X 0,Y 509.974,Z 520.955,A -85,B 0,C 180,E1 -5574.464,E2 -5574.464} C_VEL
LIN {X 0,Y 510.045,Z 520.952,A -85,B 0,C 180,E1 -5577.63,E2 -5577.63} C_VEL
LIN {X 0,Y 510.055,Z 520.947,A -85,B 0,C 180,E1 -5580.789,E2 -5580.789} C_VEL
LIN {X 0,Y 509.95,Z 520.964,A -85,B 0,C 180,E1 -5583.16,E2 -5583.16} C_VEL
LIN {X 0,Y 509.967,Z 520.957,A -85,B 0,C 180,E1 -5586.329,E2 -5586.329} C_VEL
LIN {X 0,Y 509.908,Z 520.965,A -85,B 0,C 180,E1 -5588.72,E2 -5588.72} C_VEL
LIN {X 0,Y 509.939,Z 520.963,A -85,B 0,C 180,E1 -5591.93,E2 -5591.93} C_VEL
LIN {X 0,Y 509.881,Z 520.976,A -85,B 0,C 180,E1 -5595.242,E2 -5595.242} C_VEL
LIN {X 0,Y 509.876,Z 520.971,A -85,B 0,C 180,E1 -5598.001,E2 -5598.001} C_VEL
LIN {X 0,Y 509.839,Z 520.977,A -85,B 0,C 180,E1 -5601.002,E2 -5601.002} C_VEL
LIN {X 0,Y 509.824,Z 520.982,A -85,B 0,C 180,E1 -5603.563,E2 -5603.563} C_VEL
LIN {X 0,Y 509.902,Z 520.968,A -85,B 0,C 180,E1 -5606.379,E2 -5606.379} C_VEL
LIN {X 0,Y 509.887,Z 521.047,A -85,B 0,C 180,E1 -5609.069,E2 -5609.069} C_VEL
LIN {X 0,Y 510.839,Z 527.339,A -85,B 0,C 180,E1 -5610.38,E2 -5610.38} C_VEL
LIN {X 0,Y 510.387,Z 542.677,A -85,B 0,C 180,E1 -5613.421,E2 -5613.421} C_VEL
LIN {X 0,Y 510.225,Z 548.048,A -85,B 0,C 180,E1 -5614.474,E2 -5614.474} C_VEL
LIN {X 0,Y 512.227,Z 559.207,A -85,B 0,C 180,E1 -5614.708,E2 -5614.708} C_VEL
LIN {X 0,Y 511.707,Z 654.633,A -85,B 0,C 180,E1 -5616.076,E2 -5616.076} C_VEL
LIN {X 0,Y 511.523,Z 667.93,A -85,B 0,C 180,E1 -5616.426,E2 -5616.426} C_VEL
LIN {X 0,Y 511.238,Z 680.309,A -85,B 0,C 180,E1 -5616.91,E2 -5616.91} C_VEL
LIN {X 0,Y 511.092,Z 686.554,A -85,B 0,C 180,E1 -5617.22,E2 -5617.22} C_VEL
LIN {X 0,Y 510.228,Z 691.853,A -85,B 0,C 180,E1 -5617.498,E2 -5617.498} C_VEL
LIN {X 0,Y 507.222,Z 700.264,A -85,B 0,C 180,E1 -5617.982,E2 -5617.982} C_VEL
LIN {X 0,Y 504.222,Z 708.26,A -85,B 0,C 180,E1 -5618.547,E2 -5618.547} C_VEL
LIN {X 0,Y 503.374,Z 712.897,A -85,B 0,C 180,E1 -5618.949,E2 -5618.949} C_VEL
LIN {X 0,Y 502.994,Z 722.841,A -85,B 0,C 180,E1 -5619.995,E2 -5619.995} C_VEL
LIN {X 0,Y 502.746,Z 731.124,A -85,B 0,C 180,E1 -5621.073,E2 -5621.073} C_VEL
LIN {X 0,Y 502.437,Z 738.096,A -85,B 0,C 180,E1 -5622.176,E2 -5622.176} C_VEL
LIN {X 0,Y 502.311,Z 745.032,A -85,B 0,C 180,E1 -5623.555,E2 -5623.555} C_VEL
LIN {X 0,Y 502.169,Z 750.672,A -85,B 0,C 180,E1 -5625.031,E2 -5625.031} C_VEL
LIN {X 0,Y 502.097,Z 753.841,A -85,B 0,C 180,E1 -5626.145,E2 -5626.145} C_VEL
LIN {X 0,Y 502.073,Z 755.121,A -85,B 0,C 180,E1 -5626.709,E2 -5626.709} C_VEL
LIN {X 0,Y 501.989,Z 757.145,A -85,B 0,C 180,E1 -5627.903,E2 -5627.903} C_VEL
LIN {X 0,Y 501.943,Z 758.286,A -85,B 0,C 180,E1 -5629.12,E2 -5629.12} C_VEL
LIN {X 0,Y 501.964,Z 758.514,A -85,B 0,C 180,E1 -5630.358,E2 -5630.358} C_VEL
LIN {X 0,Y 501.978,Z 757.417,A -85,B 0,C 180,E1 -5631.975,E2 -5631.975} C_VEL
LIN {X 0,Y 502.05,Z 754.864,A -85,B 0,C 180,E1 -5633.493,E2 -5633.493} C_VEL
LIN {X 0,Y 502.12,Z 750.903,A -85,B 0,C 180,E1 -5634.982,E2 -5634.982} C_VEL
LIN {X 0,Y 502.284,Z 745.373,A -85,B 0,C 180,E1 -5636.45,E2 -5636.45} C_VEL
LIN {X 0,Y 502.469,Z 739.285,A -85,B 0,C 180,E1 -5637.693,E2 -5637.693} C_VEL
LIN {X 0,Y 502.682,Z 732.229,A -85,B 0,C 180,E1 -5638.851,E2 -5638.851} C_VEL
LIN {X 0,Y 502.97,Z 723.307,A -85,B 0,C 180,E1 -5640.033,E2 -5640.033} C_VEL
LIN {X 0,Y 503.285,Z 713.518,A -85,B 0,C 180,E1 -5641.079,E2 -5641.079} C_VEL
LIN {X 0,Y 503.675,Z 702.521,A -85,B 0,C 180,E1 -5642.02,E2 -5642.02} C_VEL
LIN {X 0,Y 504.033,Z 691.735,A -85,B 0,C 180,E1 -5642.757,E2 -5642.757} C_VEL
LIN {X 0,Y 504.351,Z 679.795,A -85,B 0,C 180,E1 -5643.389,E2 -5643.389} C_VEL
LIN {X 0,Y 504.617,Z 666.302,A -85,B 0,C 180,E1 -5643.91,E2 -5643.91} C_VEL
LIN {X 0,Y 504.872,Z 653.417,A -85,B 0,C 180,E1 -5644.229,E2 -5644.229} C_VEL
LIN {X 0,Y 505.345,Z 559.791,A -85,B 0,C 180,E1 -5645.589,E2 -5645.589} C_VEL
LIN {X 0,Y 503.22,Z 548.135,A -85,B 0,C 180,E1 -5645.836,E2 -5645.836} C_VEL
LIN {X 0,Y 503.594,Z 534.674,A -85,B 0,C 180,E1 -5648.512,E2 -5648.512} C_VEL
LIN {X 0,Y 503.747,Z 527.183,A -85,B 0,C 180,E1 -5650.014,E2 -5650.014} C_VEL
LIN {X 0,Y 502.843,Z 521.851,A -85,B 0,C 180,E1 -5651.144,E2 -5651.144} C_VEL
LIN {X 0,Y 502.817,Z 521.85,A -85,B 0,C 180,E1 -5653.768,E2 -5653.768} C_VEL
LIN {X 0,Y 502.831,Z 521.849,A -85,B 0,C 180,E1 -5656.256,E2 -5656.256} C_VEL
LIN {X 0,Y 502.873,Z 521.847,A -85,B 0,C 180,E1 -5658.718,E2 -5658.718} C_VEL
LIN {X 0,Y 502.898,Z 521.836,A -85,B 0,C 180,E1 -5661.968,E2 -5661.968} C_VEL
LIN {X 0,Y 502.931,Z 521.835,A -85,B 0,C 180,E1 -5664.388,E2 -5664.388} C_VEL
LIN {X 0,Y 503.023,Z 521.822,A -85,B 0,C 180,E1 -5667.599,E2 -5667.599} C_VEL
LIN {X 0,Y 503.025,Z 521.82,A -85,B 0,C 180,E1 -5670.001,E2 -5670.001} C_VEL
LIN {X 0,Y 503.023,Z 521.823,A -85,B 0,C 180,E1 -5672.403,E2 -5672.403} C_VEL
LIN {X 0,Y 502.931,Z 521.833,A -85,B 0,C 180,E1 -5675.615,E2 -5675.615} C_VEL
LIN {X 0,Y 502.9,Z 521.836,A -85,B 0,C 180,E1 -5678.034,E2 -5678.034} C_VEL
LIN {X 0,Y 502.876,Z 521.844,A -85,B 0,C 180,E1 -5681.284,E2 -5681.284} C_VEL
LIN {X 0,Y 502.844,Z 521.845,A -85,B 0,C 180,E1 -5684.572,E2 -5684.572} C_VEL
LIN {X 0,Y 502.822,Z 521.846,A -85,B 0,C 180,E1 -5687.909,E2 -5687.909} C_VEL
LIN {X 0,Y 502.829,Z 521.846,A -85,B 0,C 180,E1 -5690.537,E2 -5690.537} C_VEL
LIN {X 0,Y 502.788,Z 521.858,A -85,B 0,C 180,E1 -5693.042,E2 -5693.042} C_VEL
LIN {X 0,Y 502.838,Z 521.846,A -85,B 0,C 180,E1 -5695.677,E2 -5695.677} C_VEL
LIN {X 0,Y 502.841,Z 521.844,A -85,B 0,C 180,E1 -5698.374,E2 -5698.374} C_VEL
LIN {X 0,Y 502.794,Z 521.854,A -85,B 0,C 180,E1 -5701.5,E2 -5701.5} C_VEL
LIN {X 0,Y 502.805,Z 521.849,A -85,B 0,C 180,E1 -5703.995,E2 -5703.995} C_VEL
LIN {X 0,Y 502.779,Z 521.859,A -85,B 0,C 180,E1 -5707.179,E2 -5707.179} C_VEL
LIN {X 0,Y 502.791,Z 521.851,A -85,B 0,C 180,E1 -5710.016,E2 -5710.016} C_VEL
LIN {X 0,Y 502.806,Z 521.848,A -85,B 0,C 180,E1 -5712.2,E2 -5712.2} C_VEL
LIN {X 0,Y 502.803,Z 521.856,A -85,B 0,C 180,E1 -5715.469,E2 -5715.469} C_VEL
LIN {X 0,Y 502.823,Z 521.848,A -85,B 0,C 180,E1 -5718.935,E2 -5718.935} C_VEL
LIN {X 0,Y 502.797,Z 521.85,A -85,B 0,C 180,E1 -5722.047,E2 -5722.047} C_VEL
LIN {X 0,Y 502.803,Z 521.851,A -85,B 0,C 180,E1 -5725.035,E2 -5725.035} C_VEL
LIN {X 0,Y 502.789,Z 521.853,A -85,B 0,C 180,E1 -5727.916,E2 -5727.916} C_VEL
LIN {X 0,Y 502.828,Z 521.845,A -85,B 0,C 180,E1 -5730.713,E2 -5730.713} C_VEL
LIN {X 0,Y 502.867,Z 521.848,A -85,B 0,C 180,E1 -5733.44,E2 -5733.44} C_VEL
LIN {X 0,Y 502.79,Z 521.852,A -85,B 0,C 180,E1 -5736.087,E2 -5736.087} C_VEL
LIN {X 0,Y 502.788,Z 521.85,A -85,B 0,C 180,E1 -5738.69,E2 -5738.69} C_VEL
LIN {X 0,Y 502.832,Z 521.848,A -85,B 0,C 180,E1 -5741.249,E2 -5741.249} C_VEL
LIN {X 0,Y 502.855,Z 521.842,A -85,B 0,C 180,E1 -5744.601,E2 -5744.601} C_VEL
LIN {X 0,Y 502.882,Z 521.843,A -85,B 0,C 180,E1 -5748.04,E2 -5748.04} C_VEL
LIN {X 0,Y 502.876,Z 521.841,A -85,B 0,C 180,E1 -5751.157,E2 -5751.157} C_VEL
LIN {X 0,Y 502.918,Z 521.84,A -85,B 0,C 180,E1 -5753.582,E2 -5753.582} C_VEL
LIN {X 0,Y 502.903,Z 521.836,A -85,B 0,C 180,E1 -5756.796,E2 -5756.796} C_VEL
LIN {X 0,Y 503.04,Z 521.82,A -85,B 0,C 180,E1 -5759.2,E2 -5759.2} C_VEL
LIN {X 0,Y 502.907,Z 521.841,A -85,B 0,C 180,E1 -5761.602,E2 -5761.602} C_VEL
LIN {X 0,Y 502.903,Z 521.837,A -85,B 0,C 180,E1 -5763.205,E2 -5763.205} C_VEL
LIN {X 0,Y 502.935,Z 521.834,A -85,B 0,C 180,E1 -5766.419,E2 -5766.419} C_VEL
LIN {X 0,Y 502.877,Z 521.839,A -85,B 0,C 180,E1 -5768.844,E2 -5768.844} C_VEL
LIN {X 0,Y 502.854,Z 521.849,A -85,B 0,C 180,E1 -5772.102,E2 -5772.102} C_VEL
LIN {X 0,Y 502.856,Z 521.843,A -85,B 0,C 180,E1 -5775.4,E2 -5775.4} C_VEL
LIN {X 0,Y 502.834,Z 521.845,A -85,B 0,C 180,E1 -5778.752,E2 -5778.752} C_VEL
LIN {X 0,Y 502.791,Z 521.85,A -85,B 0,C 180,E1 -5781.311,E2 -5781.311} C_VEL
LIN {X 0,Y 502.784,Z 521.857,A -85,B 0,C 180,E1 -5783.915,E2 -5783.915} C_VEL
LIN {X 0,Y 502.872,Z 521.842,A -85,B 0,C 180,E1 -5786.566,E2 -5786.566} C_VEL
LIN {X 0,Y 502.831,Z 521.845,A -85,B 0,C 180,E1 -5789.288,E2 -5789.288} C_VEL
LIN {X 0,Y 502.79,Z 521.858,A -85,B 0,C 180,E1 -5792.085,E2 -5792.085} C_VEL
LIN {X 0,Y 502.81,Z 521.848,A -85,B 0,C 180,E1 -5794.965,E2 -5794.965} C_VEL
LIN {X 0,Y 502.801,Z 521.854,A -85,B 0,C 180,E1 -5797.954,E2 -5797.954} C_VEL
LIN {X 0,Y 502.807,Z 521.848,A -85,B 0,C 180,E1 -5801.068,E2 -5801.068} C_VEL
LIN {X 0,Y 502.786,Z 521.859,A -85,B 0,C 180,E1 -5804.34,E2 -5804.34} C_VEL
LIN {X 0,Y 502.78,Z 521.854,A -85,B 0,C 180,E1 -5806.768,E2 -5806.768} C_VEL
LIN {X 0,Y 502.826,Z 521.846,A -85,B 0,C 180,E1 -5809.005,E2 -5809.005} C_VEL
LIN {X 0,Y 502.8,Z 521.853,A -85,B 0,C 180,E1 -5812.046,E2 -5812.046} C_VEL
LIN {X 0,Y 502.806,Z 521.849,A -85,B 0,C 180,E1 -5815.034,E2 -5815.034} C_VEL
LIN {X 0,Y 502.791,Z 521.852,A -85,B 0,C 180,E1 -5817.915,E2 -5817.915} C_VEL
LIN {X 0,Y 502.831,Z 521.851,A -85,B 0,C 180,E1 -5820.712,E2 -5820.712} C_VEL
LIN {X 0,Y 502.87,Z 521.842,A -85,B 0,C 180,E1 -5823.439,E2 -5823.439} C_VEL
LIN {X 0,Y 502.883,Z 521.865,A -85,B 0,C 180,E1 -5825.211,E2 -5825.211} C_VEL
LIN {X 0,Y 504.644,Z 532.022,A -85,B 0,C 180,E1 -5827.048,E2 -5827.048} C_VEL
LIN {X 0,Y 504.074,Z 549.762,A -85,B 0,C 180,E1 -5830.025,E2 -5830.025} C_VEL
LIN {X 0,Y 503.558,Z 566.224,A -85,B 0,C 180,E1 -5832.747,E2 -5832.747} C_VEL
LIN {X 0,Y 503.322,Z 575.052,A -85,B 0,C 180,E1 -5834.197,E2 -5834.197} C_VEL
LIN {X 0,Y 505.398,Z 588.818,A -85,B 0,C 180,E1 -5834.47,E2 -5834.47} C_VEL
LIN {X 0,Y 504.844,Z 683.485,A -85,B 0,C 180,E1 -5835.847,E2 -5835.847} C_VEL
LIN {X 0,Y 504.528,Z 696.641,A -85,B 0,C 180,E1 -5836.198,E2 -5836.198} C_VEL
LIN {X 0,Y 504.276,Z 709.321,A -85,B 0,C 180,E1 -5836.704,E2 -5836.704} C_VEL
LIN {X 0,Y 503.884,Z 721.605,A -85,B 0,C 180,E1 -5837.374,E2 -5837.374} C_VEL
LIN {X 0,Y 503.575,Z 733.555,A -85,B 0,C 180,E1 -5838.222,E2 -5838.222} C_VEL
LIN {X 0,Y 503.205,Z 743.808,A -85,B 0,C 180,E1 -5839.131,E2 -5839.131} C_VEL
LIN {X 0,Y 502.878,Z 753.021,A -85,B 0,C 180,E1 -5840.141,E2 -5840.141} C_VEL
LIN {X 0,Y 502.603,Z 761.991,A -85,B 0,C 180,E1 -5841.353,E2 -5841.353} C_VEL
LIN {X 0,Y 502.362,Z 769.21,A -85,B 0,C 180,E1 -5842.564,E2 -5842.564} C_VEL
LIN {X 0,Y 502.237,Z 774.081,A -85,B 0,C 180,E1 -5843.571,E2 -5843.571} C_VEL
LIN {X 0,Y 502.183,Z 778.816,A -85,B 0,C 180,E1 -5844.78,E2 -5844.78} C_VEL
LIN {X 0,Y 502.144,Z 782.433,A -85,B 0,C 180,E1 -5845.986,E2 -5845.986} C_VEL
LIN {X 0,Y 502.121,Z 784.298,A -85,B 0,C 180,E1 -5846.789,E2 -5846.789} C_VEL
LIN {X 0,Y 502.091,Z 785.696,A -85,B 0,C 180,E1 -5847.592,E2 -5847.592} C_VEL
LIN {X 0,Y 501.991,Z 787.299,A -85,B 0,C 180,E1 -5849.197,E2 -5849.197} C_VEL
LIN {X 0,Y 501.98,Z 787.515,A -85,B 0,C 180,E1 -5849.999,E2 -5849.999} C_VEL
LIN {X 0,Y 502.036,Z 786.691,A -85,B 0,C 180,E1 -5851.603,E2 -5851.603} C_VEL
LIN {X 0,Y 502.091,Z 785.694,A -85,B 0,C 180,E1 -5852.406,E2 -5852.406} C_VEL
LIN {X 0,Y 502.121,Z 784.294,A -85,B 0,C 180,E1 -5853.208,E2 -5853.208} C_VEL
LIN {X 0,Y 502.112,Z 781.349,A -85,B 0,C 180,E1 -5854.414,E2 -5854.414} C_VEL
LIN {X 0,Y 502.242,Z 777.366,A -85,B 0,C 180,E1 -5855.62,E2 -5855.62} C_VEL
LIN {X 0,Y 502.331,Z 771.336,A -85,B 0,C 180,E1 -5857.01,E2 -5857.01} C_VEL
LIN {X 0,Y 502.498,Z 764.535,A -85,B 0,C 180,E1 -5858.241,E2 -5858.241} C_VEL
LIN {X 0,Y 502.757,Z 756.218,A -85,B 0,C 180,E1 -5859.453,E2 -5859.453} C_VEL
LIN {X 0,Y 503.001,Z 747.685,A -85,B 0,C 180,E1 -5860.464,E2 -5860.464} C_VEL
LIN {X 0,Y 503.445,Z 737.147,A -85,B 0,C 180,E1 -5861.473,E2 -5861.473} C_VEL
LIN {X 0,Y 503.768,Z 726.122,A -85,B 0,C 180,E1 -5862.324,E2 -5862.324} C_VEL
LIN {X 0,Y 504.118,Z 715.257,A -85,B 0,C 180,E1 -5862.99,E2 -5862.99} C_VEL
LIN {X 0,Y 504.388,Z 703.436,A -85,B 0,C 180,E1 -5863.547,E2 -5863.547} C_VEL
LIN {X 0,Y 504.705,Z 689.809,A -85,B 0,C 180,E1 -5864,E2 -5864} C_VEL
LIN {X 0,Y 504.902,Z 675.985,A -85,B 0,C 180,E1 -5864.277,E2 -5864.277} C_VEL
LIN {X 0,Y 505.36,Z 587.679,A -85,B 0,C 180,E1 -5865.546,E2 -5865.546} C_VEL
LIN {X 0,Y 503.32,Z 574.753,A -85,B 0,C 180,E1 -5865.825,E2 -5865.825} C_VEL
LIN {X 0,Y 503.903,Z 554.604,A -85,B 0,C 180,E1 -5869.131,E2 -5869.131} C_VEL
LIN {X 0,Y 504.498,Z 535.573,A -85,B 0,C 180,E1 -5872.308,E2 -5872.308} C_VEL
LIN {X 0,Y 504.492,Z 530.6,A -85,B 0,C 180,E1 -5873.156,E2 -5873.156} C_VEL
LIN {X 0,Y 502.837,Z 521.852,A -85,B 0,C 180,E1 -5874.753,E2 -5874.753} C_VEL
LIN {X 0,Y 502.832,Z 521.854,A -85,B 0,C 180,E1 -5877.465,E2 -5877.465} C_VEL
LIN {X 0,Y 502.807,Z 521.853,A -85,B 0,C 180,E1 -5880.21,E2 -5880.21} C_VEL
LIN {X 0,Y 502.829,Z 521.85,A -85,B 0,C 180,E1 -5883.03,E2 -5883.03} C_VEL
LIN {X 0,Y 502.777,Z 521.856,A -85,B 0,C 180,E1 -5885.949,E2 -5885.949} C_VEL
LIN {X 0,Y 502.813,Z 521.852,A -85,B 0,C 180,E1 -5888.973,E2 -5888.973} C_VEL
LIN {X 0,Y 502.797,Z 521.852,A -85,B 0,C 180,E1 -5892.198,E2 -5892.198} C_VEL
LIN {X 0,Y 502.795,Z 521.859,A -85,B 0,C 180,E1 -5895.467,E2 -5895.467} C_VEL
LIN {X 0,Y 502.82,Z 521.851,A -85,B 0,C 180,E1 -5899.003,E2 -5899.003} C_VEL
LIN {X 0,Y 502.787,Z 521.851,A -85,B 0,C 180,E1 -5902.045,E2 -5902.045} C_VEL
LIN {X 0,Y 502.803,Z 521.853,A -85,B 0,C 180,E1 -5905.034,E2 -5905.034} C_VEL
LIN {X 0,Y 502.78,Z 521.854,A -85,B 0,C 180,E1 -5907.915,E2 -5907.915} C_VEL
LIN {X 0,Y 502.83,Z 521.846,A -85,B 0,C 180,E1 -5910.712,E2 -5910.712} C_VEL
LIN {X 0,Y 502.872,Z 521.846,A -85,B 0,C 180,E1 -5913.434,E2 -5913.434} C_VEL
LIN {X 0,Y 502.782,Z 521.85,A -85,B 0,C 180,E1 -5916.085,E2 -5916.085} C_VEL
LIN {X 0,Y 502.774,Z 521.853,A -85,B 0,C 180,E1 -5918.688,E2 -5918.688} C_VEL
LIN {X 0,Y 502.821,Z 521.85,A -85,B 0,C 180,E1 -5921.247,E2 -5921.247} C_VEL
LIN {X 0,Y 502.814,Z 521.849,A -85,B 0,C 180,E1 -5923.766,E2 -5923.766} C_VEL
LIN {X 0,Y 502.825,Z 521.847,A -85,B 0,C 180,E1 -5926.254,E2 -5926.254} C_VEL
LIN {X 0,Y 502.884,Z 521.837,A -85,B 0,C 180,E1 -5928.717,E2 -5928.717} C_VEL
LIN {X 0,Y 502.891,Z 521.839,A -85,B 0,C 180,E1 -5931.966,E2 -5931.966} C_VEL
LIN {X 0,Y 502.93,Z 521.833,A -85,B 0,C 180,E1 -5934.386,E2 -5934.386} C_VEL
LIN {X 0,Y 503.015,Z 521.828,A -85,B 0,C 180,E1 -5937.597,E2 -5937.597} C_VEL
LIN {X 0,Y 503.016,Z 521.825,A -85,B 0,C 180,E1 -5940,E2 -5940} C_VEL
LIN {X 0,Y 503.015,Z 521.822,A -85,B 0,C 180,E1 -5942.402,E2 -5942.402} C_VEL
LIN {X 0,Y 502.948,Z 521.838,A -85,B 0,C 180,E1 -5945.613,E2 -5945.613} C_VEL
LIN {X 0,Y 502.891,Z 521.84,A -85,B 0,C 180,E1 -5948.033,E2 -5948.033} C_VEL
LIN {X 0,Y 502.883,Z 521.847,A -85,B 0,C 180,E1 -5951.283,E2 -5951.283} C_VEL
LIN {X 0,Y 502.833,Z 521.847,A -85,B 0,C 180,E1 -5954.571,E2 -5954.571} C_VEL
LIN {X 0,Y 502.85,Z 521.847,A -85,B 0,C 180,E1 -5957.907,E2 -5957.907} C_VEL
LIN {X 0,Y 502.816,Z 521.849,A -85,B 0,C 180,E1 -5960.536,E2 -5960.536} C_VEL
LIN {X 0,Y 502.784,Z 521.857,A -85,B 0,C 180,E1 -5963.04,E2 -5963.04} C_VEL
LIN {X 0,Y 502.83,Z 521.852,A -85,B 0,C 180,E1 -5965.676,E2 -5965.676} C_VEL
LIN {X 0,Y 502.867,Z 521.961,A -85,B 0,C 180,E1 -5968.912,E2 -5968.912} C_VEL
LIN {X 0,Y 503.85,Z 527.749,A -85,B 0,C 180,E1 -5970.142,E2 -5970.142} C_VEL
LIN {X 0,Y 503.469,Z 540.706,A -85,B 0,C 180,E1 -5972.746,E2 -5972.746} C_VEL
LIN {X 0,Y 503.258,Z 548.29,A -85,B 0,C 180,E1 -5974.256,E2 -5974.256} C_VEL
LIN {X 0,Y 505.452,Z 561.275,A -85,B 0,C 180,E1 -5974.525,E2 -5974.525} C_VEL
LIN {X 0,Y 504.821,Z 655.172,A -85,B 0,C 180,E1 -5975.893,E2 -5975.893} C_VEL
LIN {X 0,Y 504.629,Z 668.134,A -85,B 0,C 180,E1 -5976.241,E2 -5976.241} C_VEL
LIN {X 0,Y 504.327,Z 680.308,A -85,B 0,C 180,E1 -5976.722,E2 -5976.722} C_VEL
LIN {X 0,Y 504.031,Z 692.34,A -85,B 0,C 180,E1 -5977.368,E2 -5977.368} C_VEL
LIN {X 0,Y 503.623,Z 703.35,A -85,B 0,C 180,E1 -5978.129,E2 -5978.129} C_VEL
LIN {X 0,Y 503.374,Z 712.897,A -85,B 0,C 180,E1 -5978.949,E2 -5978.949} C_VEL
LIN {X 0,Y 502.51,Z 717.403,A -85,B 0,C 180,E1 -5979.378,E2 -5979.378} C_VEL
LIN {X 0,Y 499.441,Z 724.398,A -85,B 0,C 180,E1 -5980.101,E2 -5980.101} C_VEL
LIN {X 0,Y 496.412,Z 730.854,A -85,B 0,C 180,E1 -5980.893,E2 -5980.893} C_VEL
LIN {X 0,Y 495.612,Z 734.453,A -85,B 0,C 180,E1 -5981.423,E2 -5981.423} C_VEL
LIN {X 0,Y 495.318,Z 741.492,A -85,B 0,C 180,E1 -5982.665,E2 -5982.665} C_VEL
LIN {X 0,Y 495.164,Z 747.699,A -85,B 0,C 180,E1 -5984.064,E2 -5984.064} C_VEL
LIN {X 0,Y 495.056,Z 751.673,A -85,B 0,C 180,E1 -5985.219,E2 -5985.219} C_VEL
LIN {X 0,Y 495.011,Z 754.746,A -85,B 0,C 180,E1 -5986.392,E2 -5986.392} C_VEL
LIN {X 0,Y 494.924,Z 756.974,A -85,B 0,C 180,E1 -5987.595,E2 -5987.595} C_VEL
LIN {X 0,Y 494.844,Z 758.55,A -85,B 0,C 180,E1 -5989.21,E2 -5989.21} C_VEL
LIN {X 0,Y 494.871,Z 758.734,A -85,B 0,C 180,E1 -5990.279,E2 -5990.279} C_VEL
LIN {X 0,Y 494.893,Z 758.254,A -85,B 0,C 180,E1 -5991.357,E2 -5991.357} C_VEL
LIN {X 0,Y 494.905,Z 756.685,A -85,B 0,C 180,E1 -5992.677,E2 -5992.677} C_VEL
LIN {X 0,Y 495.002,Z 753.961,A -85,B 0,C 180,E1 -5994.025,E2 -5994.025} C_VEL
LIN {X 0,Y 495.073,Z 749.873,A -85,B 0,C 180,E1 -5995.422,E2 -5995.422} C_VEL
LIN {X 0,Y 495.238,Z 744.193,A -85,B 0,C 180,E1 -5996.853,E2 -5996.853} C_VEL
LIN {X 0,Y 495.442,Z 737.792,A -85,B 0,C 180,E1 -5998.105,E2 -5998.105} C_VEL
LIN {X 0,Y 495.767,Z 730.071,A -85,B 0,C 180,E1 -5999.315,E2 -5999.315} C_VEL
LIN {X 0,Y 496.048,Z 720.632,A -85,B 0,C 180,E1 -6000.507,E2 -6000.507} C_VEL
LIN {X 0,Y 496.434,Z 711.29,A -85,B 0,C 180,E1 -6001.461,E2 -6001.461} C_VEL
LIN {X 0,Y 496.78,Z 701.536,A -85,B 0,C 180,E1 -6002.278,E2 -6002.278} C_VEL
LIN {X 0,Y 497.177,Z 690.068,A -85,B 0,C 180,E1 -6003.042,E2 -6003.042} C_VEL
LIN {X 0,Y 497.5,Z 677.384,A -85,B 0,C 180,E1 -6003.692,E2 -6003.692} C_VEL
LIN {X 0,Y 497.802,Z 664.451,A -85,B 0,C 180,E1 -6004.163,E2 -6004.163} C_VEL
LIN {X 0,Y 497.996,Z 651.451,A -85,B 0,C 180,E1 -6004.463,E2 -6004.463} C_VEL
LIN {X 0,Y 498.561,Z 561.088,A -85,B 0,C 180,E1 -6005.789,E2 -6005.789} C_VEL
LIN {X 0,Y 496.236,Z 548.371,A -85,B 0,C 180,E1 -6006.057,E2 -6006.057} C_VEL
LIN {X 0,Y 496.703,Z 533.518,A -85,B 0,C 180,E1 -6009.042,E2 -6009.042} C_VEL
LIN {X 0,Y 496.725,Z 528.098,A -85,B 0,C 180,E1 -6010.151,E2 -6010.151} C_VEL
LIN {X 0,Y 495.816,Z 522.726,A -85,B 0,C 180,E1 -6011.328,E2 -6011.328} C_VEL
LIN {X 0,Y 495.818,Z 522.727,A -85,B 0,C 180,E1 -6014.549,E2 -6014.549} C_VEL
LIN {X 0,Y 495.823,Z 522.718,A -85,B 0,C 180,E1 -6017.966,E2 -6017.966} C_VEL
LIN {X 0,Y 495.839,Z 522.722,A -85,B 0,C 180,E1 -6021.031,E2 -6021.031} C_VEL
LIN {X 0,Y 495.857,Z 522.715,A -85,B 0,C 180,E1 -6023.491,E2 -6023.491} C_VEL
LIN {X 0,Y 495.842,Z 522.722,A -85,B 0,C 180,E1 -6026.751,E2 -6026.751} C_VEL
LIN {X 0,Y 496.002,Z 522.7,A -85,B 0,C 180,E1 -6029.189,E2 -6029.189} C_VEL
LIN {X 0,Y 495.868,Z 522.713,A -85,B 0,C 180,E1 -6031.625,E2 -6031.625} C_VEL
LIN {X 0,Y 495.841,Z 522.72,A -85,B 0,C 180,E1 -6033.251,E2 -6033.251} C_VEL
LIN {X 0,Y 495.858,Z 522.716,A -85,B 0,C 180,E1 -6036.512,E2 -6036.512} C_VEL
LIN {X 0,Y 495.84,Z 522.724,A -85,B 0,C 180,E1 -6038.971,E2 -6038.971} C_VEL
LIN {X 0,Y 495.81,Z 522.72,A -85,B 0,C 180,E1 -6042.277,E2 -6042.277} C_VEL
LIN {X 0,Y 495.806,Z 522.722,A -85,B 0,C 180,E1 -6045.625,E2 -6045.625} C_VEL
LIN {X 0,Y 495.782,Z 522.731,A -85,B 0,C 180,E1 -6049.03,E2 -6049.03} C_VEL
LIN {X 0,Y 495.742,Z 522.73,A -85,B 0,C 180,E1 -6051.63,E2 -6051.63} C_VEL
LIN {X 0,Y 495.776,Z 522.728,A -85,B 0,C 180,E1 -6054.873,E2 -6054.873} C_VEL
LIN {X 0,Y 495.814,Z 522.725,A -85,B 0,C 180,E1 -6056.975,E2 -6056.975} C_VEL
LIN {X 0,Y 495.766,Z 522.725,A -85,B 0,C 180,E1 -6060.148,E2 -6060.148} C_VEL
LIN {X 0,Y 495.794,Z 522.731,A -85,B 0,C 180,E1 -6063.245,E2 -6063.245} C_VEL
LIN {X 0,Y 495.721,Z 522.731,A -85,B 0,C 180,E1 -6066.089,E2 -6066.089} C_VEL
LIN {X 0,Y 495.766,Z 522.727,A -85,B 0,C 180,E1 -6068.769,E2 -6068.769} C_VEL
LIN {X 0,Y 495.78,Z 522.726,A -85,B 0,C 180,E1 -6071.78,E2 -6071.78} C_VEL
LIN {X 0,Y 495.752,Z 522.732,A -85,B 0,C 180,E1 -6075.14,E2 -6075.14} C_VEL
LIN {X 0,Y 495.759,Z 522.726,A -85,B 0,C 180,E1 -6078.22,E2 -6078.22} C_VEL
LIN {X 0,Y 495.754,Z 522.735,A -85,B 0,C 180,E1 -6081.409,E2 -6081.409} C_VEL
LIN {X 0,Y 495.752,Z 522.727,A -85,B 0,C 180,E1 -6084.463,E2 -6084.463} C_VEL
LIN {X 0,Y 495.772,Z 522.732,A -85,B 0,C 180,E1 -6087.407,E2 -6087.407} C_VEL
LIN {X 0,Y 495.77,Z 522.725,A -85,B 0,C 180,E1 -6090.254,E2 -6090.254} C_VEL
LIN {X 0,Y 495.828,Z 522.722,A -85,B 0,C 180,E1 -6093.252,E2 -6093.252} C_VEL
LIN {X 0,Y 495.753,Z 522.733,A -85,B 0,C 180,E1 -6095.726,E2 -6095.726} C_VEL
LIN {X 0,Y 495.747,Z 522.728,A -85,B 0,C 180,E1 -6098.372,E2 -6098.372} C_VEL
LIN {X 0,Y 495.787,Z 522.723,A -85,B 0,C 180,E1 -6100.972,E2 -6100.972} C_VEL
LIN {X 0,Y 495.813,Z 522.72,A -85,B 0,C 180,E1 -6104.377,E2 -6104.377} C_VEL
LIN {X 0,Y 495.789,Z 522.722,A -85,B 0,C 180,E1 -6106.891,E2 -6106.891} C_VEL
LIN {X 0,Y 495.779,Z 522.727,A -85,B 0,C 180,E1 -6109.381,E2 -6109.381} C_VEL
LIN {X 0,Y 495.878,Z 522.718,A -85,B 0,C 180,E1 -6111.853,E2 -6111.853} C_VEL
LIN {X 0,Y 495.898,Z 522.71,A -85,B 0,C 180,E1 -6114.307,E2 -6114.307} C_VEL
LIN {X 0,Y 495.999,Z 522.701,A -85,B 0,C 180,E1 -6117.564,E2 -6117.564} C_VEL
LIN {X 0,Y 495.99,Z 522.697,A -85,B 0,C 180,E1 -6120.812,E2 -6120.812} C_VEL
LIN {X 0,Y 496,Z 522.697,A -85,B 0,C 180,E1 -6122.437,E2 -6122.437} C_VEL
LIN {X 0,Y 495.902,Z 522.714,A -85,B 0,C 180,E1 -6125.694,E2 -6125.694} C_VEL
LIN {X 0,Y 495.879,Z 522.716,A -85,B 0,C 180,E1 -6128.148,E2 -6128.148} C_VEL
LIN {X 0,Y 495.859,Z 522.716,A -85,B 0,C 180,E1 -6131.445,E2 -6131.445} C_VEL
LIN {X 0,Y 495.798,Z 522.721,A -85,B 0,C 180,E1 -6134.783,E2 -6134.783} C_VEL
LIN {X 0,Y 495.772,Z 522.725,A -85,B 0,C 180,E1 -6137.32,E2 -6137.32} C_VEL
LIN {X 0,Y 495.779,Z 522.73,A -85,B 0,C 180,E1 -6139.89,E2 -6139.89} C_VEL
LIN {X 0,Y 495.766,Z 522.725,A -85,B 0,C 180,E1 -6142.86,E2 -6142.86} C_VEL
LIN {X 0,Y 495.789,Z 522.731,A -85,B 0,C 180,E1 -6146.068,E2 -6146.068} C_VEL
LIN {X 0,Y 495.778,Z 522.724,A -85,B 0,C 180,E1 -6148.815,E2 -6148.815} C_VEL
LIN {X 0,Y 495.762,Z 522.728,A -85,B 0,C 180,E1 -6151.725,E2 -6151.725} C_VEL
LIN {X 0,Y 495.774,Z 522.726,A -85,B 0,C 180,E1 -6154.693,E2 -6154.693} C_VEL
LIN {X 0,Y 495.738,Z 522.729,A -85,B 0,C 180,E1 -6157.561,E2 -6157.561} C_VEL
LIN {X 0,Y 495.761,Z 522.728,A -85,B 0,C 180,E1 -6160.701,E2 -6160.701} C_VEL
LIN {X 0,Y 495.724,Z 522.732,A -85,B 0,C 180,E1 -6163.693,E2 -6163.693} C_VEL
LIN {X 0,Y 495.733,Z 522.738,A -85,B 0,C 180,E1 -6166.305,E2 -6166.305} C_VEL
LIN {X 0,Y 495.773,Z 522.724,A -85,B 0,C 180,E1 -6169.3,E2 -6169.3} C_VEL
LIN {X 0,Y 495.736,Z 522.737,A -85,B 0,C 180,E1 -6172.438,E2 -6172.438} C_VEL
LIN {X 0,Y 495.785,Z 522.722,A -85,B 0,C 180,E1 -6175.456,E2 -6175.456} C_VEL
LIN {X 0,Y 495.763,Z 522.734,A -85,B 0,C 180,E1 -6178.363,E2 -6178.363} C_VEL
LIN {X 0,Y 495.794,Z 522.723,A -85,B 0,C 180,E1 -6181.506,E2 -6181.506} C_VEL
LIN {X 0,Y 495.798,Z 522.726,A -85,B 0,C 180,E1 -6183.931,E2 -6183.931} C_VEL
LIN {X 0,Y 495.834,Z 522.754,A -85,B 0,C 180,E1 -6185.02,E2 -6185.02} C_VEL
LIN {X 0,Y 497.69,Z 533.134,A -85,B 0,C 180,E1 -6186.928,E2 -6186.928} C_VEL
LIN {X 0,Y 497.17,Z 548.319,A -85,B 0,C 180,E1 -6189.52,E2 -6189.52} C_VEL
LIN {X 0,Y 496.576,Z 566.028,A -85,B 0,C 180,E1 -6192.496,E2 -6192.496} C_VEL
LIN {X 0,Y 496.33,Z 574.832,A -85,B 0,C 180,E1 -6193.964,E2 -6193.964} C_VEL
LIN {X 0,Y 498.555,Z 589.704,A -85,B 0,C 180,E1 -6194.267,E2 -6194.267} C_VEL
LIN {X 0,Y 497.962,Z 683.111,A -85,B 0,C 180,E1 -6195.647,E2 -6195.647} C_VEL
LIN {X 0,Y 497.642,Z 696.321,A -85,B 0,C 180,E1 -6196.003,E2 -6196.003} C_VEL
LIN {X 0,Y 497.351,Z 709.03,A -85,B 0,C 180,E1 -6196.516,E2 -6196.516} C_VEL
LIN {X 0,Y 496.94,Z 721.372,A -85,B 0,C 180,E1 -6197.197,E2 -6197.197} C_VEL
LIN {X 0,Y 496.593,Z 733.304,A -85,B 0,C 180,E1 -6198.054,E2 -6198.054} C_VEL
LIN {X 0,Y 496.215,Z 743.57,A -85,B 0,C 180,E1 -6198.976,E2 -6198.976} C_VEL
LIN {X 0,Y 495.856,Z 752.791,A -85,B 0,C 180,E1 -6200,E2 -6200} C_VEL
LIN {X 0,Y 495.542,Z 761.767,A -85,B 0,C 180,E1 -6201.229,E2 -6201.229} C_VEL
LIN {X 0,Y 495.313,Z 768.993,A -85,B 0,C 180,E1 -6202.457,E2 -6202.457} C_VEL
LIN {X 0,Y 495.147,Z 774.975,A -85,B 0,C 180,E1 -6203.738,E2 -6203.738} C_VEL
LIN {X 0,Y 495.039,Z 779.922,A -85,B 0,C 180,E1 -6205.112,E2 -6205.112} C_VEL
LIN {X 0,Y 495.039,Z 782.225,A -85,B 0,C 180,E1 -6205.928,E2 -6205.928} C_VEL
LIN {X 0,Y 495.043,Z 784.093,A -85,B 0,C 180,E1 -6206.743,E2 -6206.743} C_VEL
LIN {X 0,Y 494.998,Z 785.492,A -85,B 0,C 180,E1 -6207.558,E2 -6207.558} C_VEL
LIN {X 0,Y 494.962,Z 786.489,A -85,B 0,C 180,E1 -6208.372,E2 -6208.372} C_VEL
LIN {X 0,Y 494.898,Z 787.311,A -85,B 0,C 180,E1 -6209.999,E2 -6209.999} C_VEL
LIN {X 0,Y 494.962,Z 786.485,A -85,B 0,C 180,E1 -6211.626,E2 -6211.626} C_VEL
LIN {X 0,Y 494.997,Z 785.485,A -85,B 0,C 180,E1 -6212.44,E2 -6212.44} C_VEL
LIN {X 0,Y 495.042,Z 784.084,A -85,B 0,C 180,E1 -6213.254,E2 -6213.254} C_VEL
LIN {X 0,Y 495.016,Z 781.134,A -85,B 0,C 180,E1 -6214.477,E2 -6214.477} C_VEL
LIN {X 0,Y 495.159,Z 777.146,A -85,B 0,C 180,E1 -6215.701,E2 -6215.701} C_VEL
LIN {X 0,Y 495.256,Z 771.008,A -85,B 0,C 180,E1 -6217.131,E2 -6217.131} C_VEL
LIN {X 0,Y 495.442,Z 764.299,A -85,B 0,C 180,E1 -6218.359,E2 -6218.359} C_VEL
LIN {X 0,Y 495.73,Z 755.974,A -85,B 0,C 180,E1 -6219.588,E2 -6219.588} C_VEL
LIN {X 0,Y 495.994,Z 747.43,A -85,B 0,C 180,E1 -6220.613,E2 -6220.613} C_VEL
LIN {X 0,Y 496.467,Z 736.878,A -85,B 0,C 180,E1 -6221.636,E2 -6221.636} C_VEL
LIN {X 0,Y 496.809,Z 725.84,A -85,B 0,C 180,E1 -6222.5,E2 -6222.5} C_VEL
LIN {X 0,Y 497.162,Z 714.954,A -85,B 0,C 180,E1 -6223.175,E2 -6223.175} C_VEL
LIN {X 0,Y 497.485,Z 703.099,A -85,B 0,C 180,E1 -6223.738,E2 -6223.738} C_VEL
LIN {X 0,Y 497.815,Z 689.427,A -85,B 0,C 180,E1 -6224.198,E2 -6224.198} C_VEL
LIN {X 0,Y 498.023,Z 675.46,A -85,B 0,C 180,E1 -6224.479,E2 -6224.479} C_VEL
LIN {X 0,Y 498.402,Z 587.957,A -85,B 0,C 180,E1 -6225.761,E2 -6225.761} C_VEL
LIN {X 0,Y 496.28,Z 574.636,A -85,B 0,C 180,E1 -6226.036,E2 -6226.036} C_VEL
LIN {X 0,Y 496.911,Z 555.673,A -85,B 0,C 180,E1 -6229.197,E2 -6229.197} C_VEL
LIN {X 0,Y 497.598,Z 535.391,A -85,B 0,C 180,E1 -6232.634,E2 -6232.634} C_VEL
LIN {X 0,Y 497.47,Z 531.452,A -85,B 0,C 180,E1 -6233.322,E2 -6233.322} C_VEL
LIN {X 0,Y 495.797,Z 522.729,A -85,B 0,C 180,E1 -6234.978,E2 -6234.978} C_VEL
LIN {X 0,Y 495.78,Z 522.732,A -85,B 0,C 180,E1 -6237.89,E2 -6237.89} C_VEL
LIN {X 0,Y 495.75,Z 522.732,A -85,B 0,C 180,E1 -6240.686,E2 -6240.686} C_VEL
LIN {X 0,Y 495.757,Z 522.735,A -85,B 0,C 180,E1 -6243.563,E2 -6243.563} C_VEL
LIN {X 0,Y 495.729,Z 522.732,A -85,B 0,C 180,E1 -6246.542,E2 -6246.542} C_VEL
LIN {X 0,Y 495.778,Z 522.733,A -85,B 0,C 180,E1 -6249.634,E2 -6249.634} C_VEL
LIN {X 0,Y 495.735,Z 522.732,A -85,B 0,C 180,E1 -6252.506,E2 -6252.506} C_VEL
LIN {X 0,Y 495.743,Z 522.735,A -85,B 0,C 180,E1 -6255.138,E2 -6255.138} C_VEL
LIN {X 0,Y 495.754,Z 522.729,A -85,B 0,C 180,E1 -6258.218,E2 -6258.218} C_VEL
LIN {X 0,Y 495.762,Z 522.732,A -85,B 0,C 180,E1 -6261.23,E2 -6261.23} C_VEL
LIN {X 0,Y 495.751,Z 522.728,A -85,B 0,C 180,E1 -6264.462,E2 -6264.462} C_VEL
LIN {X 0,Y 495.761,Z 522.734,A -85,B 0,C 180,E1 -6267.405,E2 -6267.405} C_VEL
LIN {X 0,Y 495.773,Z 522.725,A -85,B 0,C 180,E1 -6270.254,E2 -6270.254} C_VEL
LIN {X 0,Y 495.825,Z 522.722,A -85,B 0,C 180,E1 -6273.247,E2 -6273.247} C_VEL
LIN {X 0,Y 495.743,Z 522.73,A -85,B 0,C 180,E1 -6275.724,E2 -6275.724} C_VEL
LIN {X 0,Y 495.738,Z 522.729,A -85,B 0,C 180,E1 -6278.37,E2 -6278.37} C_VEL
LIN {X 0,Y 495.775,Z 522.724,A -85,B 0,C 180,E1 -6280.971,E2 -6280.971} C_VEL
LIN {X 0,Y 495.771,Z 522.729,A -85,B 0,C 180,E1 -6283.529,E2 -6283.529} C_VEL
LIN {X 0,Y 495.788,Z 522.724,A -85,B 0,C 180,E1 -6286.055,E2 -6286.055} C_VEL
LIN {X 0,Y 495.858,Z 522.712,A -85,B 0,C 180,E1 -6288.555,E2 -6288.555} C_VEL
LIN {X 0,Y 495.863,Z 522.715,A -85,B 0,C 180,E1 -6291.851,E2 -6291.851} C_VEL
LIN {X 0,Y 495.887,Z 522.711,A -85,B 0,C 180,E1 -6294.306,E2 -6294.306} C_VEL
LIN {X 0,Y 495.984,Z 522.704,A -85,B 0,C 180,E1 -6297.563,E2 -6297.563} C_VEL
LIN {X 0,Y 495.987,Z 522.7,A -85,B 0,C 180,E1 -6300,E2 -6300} C_VEL
LIN {X 0,Y 495.984,Z 522.698,A -85,B 0,C 180,E1 -6302.436,E2 -6302.436} C_VEL
LIN {X 0,Y 495.902,Z 522.714,A -85,B 0,C 180,E1 -6305.693,E2 -6305.693} C_VEL
LIN {X 0,Y 495.862,Z 522.715,A -85,B 0,C 180,E1 -6308.148,E2 -6308.148} C_VEL
LIN {X 0,Y 495.863,Z 522.721,A -85,B 0,C 180,E1 -6311.444,E2 -6311.444} C_VEL
LIN {X 0,Y 495.778,Z 522.728,A -85,B 0,C 180,E1 -6314.783,E2 -6314.783} C_VEL
LIN {X 0,Y 495.776,Z 522.733,A -85,B 0,C 180,E1 -6317.318,E2 -6317.318} C_VEL
LIN {X 0,Y 495.766,Z 522.73,A -85,B 0,C 180,E1 -6319.89,E2 -6319.89} C_VEL
LIN {X 0,Y 495.745,Z 522.732,A -85,B 0,C 180,E1 -6322.861,E2 -6322.861} C_VEL
LIN {X 0,Y 495.787,Z 522.727,A -85,B 0,C 180,E1 -6326.068,E2 -6326.068} C_VEL
LIN {X 0,Y 495.784,Z 522.731,A -85,B 0,C 180,E1 -6328.714,E2 -6328.714} C_VEL
LIN {X 0,Y 496.885,Z 528.793,A -85,B 0,C 180,E1 -6330.026,E2 -6330.026} C_VEL
LIN {X 0,Y 496.513,Z 541.135,A -85,B 0,C 180,E1 -6332.539,E2 -6332.539} C_VEL
LIN {X 0,Y 496.326,Z 548.761,A -85,B 0,C 180,E1 -6334.039,E2 -6334.039} C_VEL
LIN {X 0,Y 498.543,Z 560.793,A -85,B 0,C 180,E1 -6334.294,E2 -6334.294} C_VEL
LIN {X 0,Y 497.947,Z 655.383,A -85,B 0,C 180,E1 -6335.698,E2 -6335.698} C_VEL
LIN {X 0,Y 497.744,Z 668.551,A -85,B 0,C 180,E1 -6336.058,E2 -6336.058} C_VEL
LIN {X 0,Y 497.429,Z 680.205,A -85,B 0,C 180,E1 -6336.524,E2 -6336.524} C_VEL
LIN {X 0,Y 497.097,Z 692.444,A -85,B 0,C 180,E1 -6337.185,E2 -6337.185} C_VEL
LIN {X 0,Y 496.695,Z 703.016,A -85,B 0,C 180,E1 -6337.921,E2 -6337.921} C_VEL
LIN {X 0,Y 496.37,Z 713.75,A -85,B 0,C 180,E1 -6338.858,E2 -6338.858} C_VEL
LIN {X 0,Y 495.999,Z 722.92,A -85,B 0,C 180,E1 -6339.84,E2 -6339.84} C_VEL
LIN {X 0,Y 495.721,Z 731.616,A -85,B 0,C 180,E1 -6340.989,E2 -6340.989} C_VEL
LIN {X 0,Y 495.612,Z 734.453,A -85,B 0,C 180,E1 -6341.423,E2 -6341.423} C_VEL
LIN {X 0,Y 494.818,Z 737.87,A -85,B 0,C 180,E1 -6341.974,E2 -6341.974} C_VEL
LIN {X 0,Y 491.819,Z 743.014,A -85,B 0,C 180,E1 -6342.895,E2 -6342.895} C_VEL
LIN {X 0,Y 488.829,Z 747.467,A -85,B 0,C 180,E1 -6343.873,E2 -6343.873} C_VEL
LIN {X 0,Y 488.06,Z 749.8,A -85,B 0,C 180,E1 -6344.505,E2 -6344.505} C_VEL
LIN {X 0,Y 487.93,Z 754.345,A -85,B 0,C 180,E1 -6346.069,E2 -6346.069} C_VEL
LIN {X 0,Y 487.856,Z 756.928,A -85,B 0,C 180,E1 -6347.386,E2 -6347.386} C_VEL
LIN {X 0,Y 487.769,Z 758.295,A -85,B 0,C 180,E1 -6348.524,E2 -6348.524} C_VEL
LIN {X 0,Y 487.758,Z 758.936,A -85,B 0,C 180,E1 -6349.788,E2 -6349.788} C_VEL
LIN {X 0,Y 487.777,Z 758.639,A -85,B 0,C 180,E1 -6351.081,E2 -6351.081} C_VEL
LIN {X 0,Y 487.825,Z 756.8,A -85,B 0,C 180,E1 -6352.767,E2 -6352.767} C_VEL
LIN {X 0,Y 487.947,Z 753.567,A -85,B 0,C 180,E1 -6354.317,E2 -6354.317} C_VEL
LIN {X 0,Y 488.06,Z 748.899,A -85,B 0,C 180,E1 -6355.836,E2 -6355.836} C_VEL
LIN {X 0,Y 488.22,Z 743.771,A -85,B 0,C 180,E1 -6357.085,E2 -6357.085} C_VEL
LIN {X 0,Y 488.441,Z 736.598,A -85,B 0,C 180,E1 -6358.459,E2 -6358.459} C_VEL
LIN {X 0,Y 488.775,Z 729.001,A -85,B 0,C 180,E1 -6359.623,E2 -6359.623} C_VEL
LIN {X 0,Y 489.087,Z 719.95,A -85,B 0,C 180,E1 -6360.755,E2 -6360.755} C_VEL
LIN {X 0,Y 489.484,Z 710.442,A -85,B 0,C 180,E1 -6361.719,E2 -6361.719} C_VEL
LIN {X 0,Y 489.903,Z 700.23,A -85,B 0,C 180,E1 -6362.559,E2 -6362.559} C_VEL
LIN {X 0,Y 490.311,Z 688.416,A -85,B 0,C 180,E1 -6363.333,E2 -6363.333} C_VEL
LIN {X 0,Y 490.634,Z 677.165,A -85,B 0,C 180,E1 -6363.901,E2 -6363.901} C_VEL
LIN {X 0,Y 490.93,Z 664.294,A -85,B 0,C 180,E1 -6364.371,E2 -6364.371} C_VEL
LIN {X 0,Y 491.146,Z 650.852,A -85,B 0,C 180,E1 -6364.679,E2 -6364.679} C_VEL
LIN {X 0,Y 491.666,Z 561.197,A -85,B 0,C 180,E1 -6366.017,E2 -6366.017} C_VEL
LIN {X 0,Y 489.238,Z 548.467,A -85,B 0,C 180,E1 -6366.303,E2 -6366.303} C_VEL
LIN {X 0,Y 489.755,Z 534.275,A -85,B 0,C 180,E1 -6369.198,E2 -6369.198} C_VEL
LIN {X 0,Y 489.708,Z 529.012,A -85,B 0,C 180,E1 -6370.291,E2 -6370.291} C_VEL
LIN {X 0,Y 488.78,Z 523.602,A -85,B 0,C 180,E1 -6371.506,E2 -6371.506} C_VEL
LIN {X 0,Y 488.757,Z 523.606,A -85,B 0,C 180,E1 -6375.001,E2 -6375.001} C_VEL
LIN {X 0,Y 488.801,Z 523.596,A -85,B 0,C 180,E1 -6378.389,E2 -6378.389} C_VEL
LIN {X 0,Y 488.813,Z 523.591,A -85,B 0,C 180,E1 -6381.735,E2 -6381.735} C_VEL
LIN {X 0,Y 488.845,Z 523.588,A -85,B 0,C 180,E1 -6384.225,E2 -6384.225} C_VEL
LIN {X 0,Y 488.959,Z 523.574,A -85,B 0,C 180,E1 -6387.53,E2 -6387.53} C_VEL
LIN {X 0,Y 488.952,Z 523.581,A -85,B 0,C 180,E1 -6390.825,E2 -6390.825} C_VEL
LIN {X 0,Y 488.96,Z 523.575,A -85,B 0,C 180,E1 -6392.473,E2 -6392.473} C_VEL
LIN {X 0,Y 488.845,Z 523.587,A -85,B 0,C 180,E1 -6395.777,E2 -6395.777} C_VEL
LIN {X 0,Y 488.816,Z 523.591,A -85,B 0,C 180,E1 -6398.268,E2 -6398.268} C_VEL
LIN {X 0,Y 488.804,Z 523.594,A -85,B 0,C 180,E1 -6401.614,E2 -6401.614} C_VEL
LIN {X 0,Y 488.761,Z 523.606,A -85,B 0,C 180,E1 -6405.001,E2 -6405.001} C_VEL
LIN {X 0,Y 488.747,Z 523.6,A -85,B 0,C 180,E1 -6408.444,E2 -6408.444} C_VEL
LIN {X 0,Y 488.707,Z 523.612,A -85,B 0,C 180,E1 -6411.072,E2 -6411.072} C_VEL
LIN {X 0,Y 488.684,Z 523.609,A -85,B 0,C 180,E1 -6413.747,E2 -6413.747} C_VEL
LIN {X 0,Y 488.792,Z 523.599,A -85,B 0,C 180,E1 -6416.945,E2 -6416.945} C_VEL
LIN {X 0,Y 488.711,Z 523.604,A -85,B 0,C 180,E1 -6420.364,E2 -6420.364} C_VEL
LIN {X 0,Y 488.736,Z 523.606,A -85,B 0,C 180,E1 -6423.485,E2 -6423.485} C_VEL
LIN {X 0,Y 488.684,Z 523.607,A -85,B 0,C 180,E1 -6426.355,E2 -6426.355} C_VEL
LIN {X 0,Y 488.703,Z 523.613,A -85,B 0,C 180,E1 -6429.255,E2 -6429.255} C_VEL
LIN {X 0,Y 488.726,Z 523.607,A -85,B 0,C 180,E1 -6431.603,E2 -6431.603} C_VEL
LIN {X 0,Y 488.715,Z 523.605,A -85,B 0,C 180,E1 -6434.802,E2 -6434.802} C_VEL
LIN {X 0,Y 488.694,Z 523.614,A -85,B 0,C 180,E1 -6437.475,E2 -6437.475} C_VEL
LIN {X 0,Y 488.736,Z 523.606,A -85,B 0,C 180,E1 -6439.678,E2 -6439.678} C_VEL
LIN {X 0,Y 488.682,Z 523.609,A -85,B 0,C 180,E1 -6442.842,E2 -6442.842} C_VEL
LIN {X 0,Y 488.734,Z 523.604,A -85,B 0,C 180,E1 -6445.888,E2 -6445.888} C_VEL
LIN {X 0,Y 488.696,Z 523.606,A -85,B 0,C 180,E1 -6448.821,E2 -6448.821} C_VEL
LIN {X 0,Y 488.749,Z 523.606,A -85,B 0,C 180,E1 -6451.672,E2 -6451.672} C_VEL
LIN {X 0,Y 488.745,Z 523.6,A -85,B 0,C 180,E1 -6454.445,E2 -6454.445} C_VEL
LIN {X 0,Y 488.728,Z 523.604,A -85,B 0,C 180,E1 -6457.154,E2 -6457.154} C_VEL
LIN {X 0,Y 488.73,Z 523.608,A -85,B 0,C 180,E1 -6459.811,E2 -6459.811} C_VEL
LIN {X 0,Y 488.72,Z 523.603,A -85,B 0,C 180,E1 -6462.423,E2 -6462.423} C_VEL
LIN {X 0,Y 488.768,Z 523.598,A -85,B 0,C 180,E1 -6465,E2 -6465} C_VEL
LIN {X 0,Y 488.811,Z 523.592,A -85,B 0,C 180,E1 -6468.388,E2 -6468.388} C_VEL
LIN {X 0,Y 488.823,Z 523.599,A -85,B 0,C 180,E1 -6471.734,E2 -6471.734} C_VEL
LIN {X 0,Y 488.856,Z 523.588,A -85,B 0,C 180,E1 -6474.225,E2 -6474.225} C_VEL
LIN {X 0,Y 488.967,Z 523.577,A -85,B 0,C 180,E1 -6477.529,E2 -6477.529} C_VEL
LIN {X 0,Y 488.941,Z 523.575,A -85,B 0,C 180,E1 -6480.824,E2 -6480.824} C_VEL
LIN {X 0,Y 488.967,Z 523.573,A -85,B 0,C 180,E1 -6482.472,E2 -6482.472} C_VEL
LIN {X 0,Y 488.862,Z 523.592,A -85,B 0,C 180,E1 -6485.776,E2 -6485.776} C_VEL
LIN {X 0,Y 488.823,Z 523.594,A -85,B 0,C 180,E1 -6488.267,E2 -6488.267} C_VEL
LIN {X 0,Y 488.813,Z 523.595,A -85,B 0,C 180,E1 -6491.613,E2 -6491.613} C_VEL
LIN {X 0,Y 488.77,Z 523.596,A -85,B 0,C 180,E1 -6495.001,E2 -6495.001} C_VEL
LIN {X 0,Y 488.754,Z 523.601,A -85,B 0,C 180,E1 -6498.443,E2 -6498.443} C_VEL
LIN {X 0,Y 488.715,Z 523.603,A -85,B 0,C 180,E1 -6501.071,E2 -6501.071} C_VEL
LIN {X 0,Y 488.688,Z 523.611,A -85,B 0,C 180,E1 -6503.746,E2 -6503.746} C_VEL
LIN {X 0,Y 488.799,Z 523.593,A -85,B 0,C 180,E1 -6506.943,E2 -6506.943} C_VEL
LIN {X 0,Y 488.717,Z 523.608,A -85,B 0,C 180,E1 -6510.363,E2 -6510.363} C_VEL
LIN {X 0,Y 488.737,Z 523.601,A -85,B 0,C 180,E1 -6513.483,E2 -6513.483} C_VEL
LIN {X 0,Y 488.695,Z 523.612,A -85,B 0,C 180,E1 -6516.355,E2 -6516.355} C_VEL
LIN {X 0,Y 488.708,Z 523.604,A -85,B 0,C 180,E1 -6519.254,E2 -6519.254} C_VEL
LIN {X 0,Y 488.694,Z 523.611,A -85,B 0,C 180,E1 -6522.526,E2 -6522.526} C_VEL
LIN {X 0,Y 488.708,Z 523.604,A -85,B 0,C 180,E1 -6525.197,E2 -6525.197} C_VEL
LIN {X 0,Y 488.714,Z 523.611,A -85,B 0,C 180,E1 -6528.4,E2 -6528.4} C_VEL
LIN {X 0,Y 488.71,Z 523.605,A -85,B 0,C 180,E1 -6530.947,E2 -6530.947} C_VEL
LIN {X 0,Y 488.684,Z 523.609,A -85,B 0,C 180,E1 -6533.867,E2 -6533.867} C_VEL
LIN {X 0,Y 488.745,Z 523.602,A -85,B 0,C 180,E1 -6536.877,E2 -6536.877} C_VEL
LIN {X 0,Y 488.731,Z 523.604,A -85,B 0,C 180,E1 -6539.78,E2 -6539.78} C_VEL
LIN {X 0,Y 488.799,Z 523.597,A -85,B 0,C 180,E1 -6543.056,E2 -6543.056} C_VEL
LIN {X 0,Y 488.803,Z 523.766,A -85,B 0,C 180,E1 -6544.847,E2 -6544.847} C_VEL
LIN {X 0,Y 490.758,Z 534.519,A -85,B 0,C 180,E1 -6546.856,E2 -6546.856} C_VEL
LIN {X 0,Y 490.193,Z 549.402,A -85,B 0,C 180,E1 -6549.434,E2 -6549.434} C_VEL
LIN {X 0,Y 489.574,Z 567.097,A -85,B 0,C 180,E1 -6552.453,E2 -6552.453} C_VEL
LIN {X 0,Y 489.318,Z 574.671,A -85,B 0,C 180,E1 -6553.733,E2 -6553.733} C_VEL
LIN {X 0,Y 491.725,Z 591.056,A -85,B 0,C 180,E1 -6554.066,E2 -6554.066} C_VEL
LIN {X 0,Y 491.096,Z 682.737,A -85,B 0,C 180,E1 -6555.442,E2 -6555.442} C_VEL
LIN {X 0,Y 490.763,Z 696.001,A -85,B 0,C 180,E1 -6555.803,E2 -6555.803} C_VEL
LIN {X 0,Y 490.423,Z 708.739,A -85,B 0,C 180,E1 -6556.322,E2 -6556.322} C_VEL
LIN {X 0,Y 490.026,Z 719.978,A -85,B 0,C 180,E1 -6556.938,E2 -6556.938} C_VEL
LIN {X 0,Y 489.625,Z 731.754,A -85,B 0,C 180,E1 -6557.776,E2 -6557.776} C_VEL
LIN {X 0,Y 489.25,Z 742.268,A -85,B 0,C 180,E1 -6558.712,E2 -6558.712} C_VEL
LIN {X 0,Y 488.862,Z 750.861,A -85,B 0,C 180,E1 -6559.646,E2 -6559.646} C_VEL
LIN {X 0,Y 488.571,Z 758.788,A -85,B 0,C 180,E1 -6560.686,E2 -6560.686} C_VEL
LIN {X 0,Y 488.329,Z 766.53,A -85,B 0,C 180,E1 -6561.932,E2 -6561.932} C_VEL
LIN {X 0,Y 488.102,Z 773.654,A -85,B 0,C 180,E1 -6563.384,E2 -6563.384} C_VEL
LIN {X 0,Y 488.034,Z 778.397,A -85,B 0,C 180,E1 -6564.628,E2 -6564.628} C_VEL
LIN {X 0,Y 487.935,Z 782.018,A -85,B 0,C 180,E1 -6565.869,E2 -6565.869} C_VEL
LIN {X 0,Y 487.966,Z 783.888,A -85,B 0,C 180,E1 -6566.696,E2 -6566.696} C_VEL
LIN {X 0,Y 487.909,Z 785.287,A -85,B 0,C 180,E1 -6567.522,E2 -6567.522} C_VEL
LIN {X 0,Y 487.891,Z 786.285,A -85,B 0,C 180,E1 -6568.348,E2 -6568.348} C_VEL
LIN {X 0,Y 487.819,Z 787.107,A -85,B 0,C 180,E1 -6569.999,E2 -6569.999} C_VEL
LIN {X 0,Y 487.891,Z 786.279,A -85,B 0,C 180,E1 -6571.65,E2 -6571.65} C_VEL
LIN {X 0,Y 487.908,Z 785.277,A -85,B 0,C 180,E1 -6572.475,E2 -6572.475} C_VEL
LIN {X 0,Y 487.965,Z 783.873,A -85,B 0,C 180,E1 -6573.301,E2 -6573.301} C_VEL
LIN {X 0,Y 487.927,Z 780.919,A -85,B 0,C 180,E1 -6574.543,E2 -6574.543} C_VEL
LIN {X 0,Y 488.058,Z 776.926,A -85,B 0,C 180,E1 -6575.784,E2 -6575.784} C_VEL
LIN {X 0,Y 488.183,Z 770.78,A -85,B 0,C 180,E1 -6577.235,E2 -6577.235} C_VEL
LIN {X 0,Y 488.376,Z 764.063,A -85,B 0,C 180,E1 -6578.481,E2 -6578.481} C_VEL
LIN {X 0,Y 488.697,Z 755.73,A -85,B 0,C 180,E1 -6579.727,E2 -6579.727} C_VEL
LIN {X 0,Y 489.004,Z 747.175,A -85,B 0,C 180,E1 -6580.767,E2 -6580.767} C_VEL
LIN {X 0,Y 489.487,Z 736.609,A -85,B 0,C 180,E1 -6581.805,E2 -6581.805} C_VEL
LIN {X 0,Y 489.889,Z 724.986,A -85,B 0,C 180,E1 -6582.721,E2 -6582.721} C_VEL
LIN {X 0,Y 490.263,Z 712.676,A -85,B 0,C 180,E1 -6583.469,E2 -6583.469} C_VEL
LIN {X 0,Y 490.68,Z 700.158,A -85,B 0,C 180,E1 -6584.038,E2 -6584.038} C_VEL
LIN {X 0,Y 490.978,Z 687.102,A -85,B 0,C 180,E1 -6584.453,E2 -6584.453} C_VEL
LIN {X 0,Y 491.187,Z 671.398,A -85,B 0,C 180,E1 -6584.738,E2 -6584.738} C_VEL
LIN {X 0,Y 491.599,Z 588.99,A -85,B 0,C 180,E1 -6585.966,E2 -6585.966} C_VEL
LIN {X 0,Y 489.335,Z 574.332,A -85,B 0,C 180,E1 -6586.284,E2 -6586.284} C_VEL
LIN {X 0,Y 489.916,Z 555.473,A -85,B 0,C 180,E1 -6589.482,E2 -6589.482} C_VEL
LIN {X 0,Y 490.645,Z 537.748,A -85,B 0,C 180,E1 -6592.529,E2 -6592.529} C_VEL
LIN {X 0,Y 490.743,Z 534.261,A -85,B 0,C 180,E1 -6593.138,E2 -6593.138} C_VEL
LIN {X 0,Y 488.769,Z 523.605,A -85,B 0,C 180,E1 -6595.149,E2 -6595.149} C_VEL
LIN {X 0,Y 488.745,Z 523.609,A -85,B 0,C 180,E1 -6597.395,E2 -6597.395} C_VEL
LIN {X 0,Y 488.707,Z 523.609,A -85,B 0,C 180,E1 -6600.362,E2 -6600.362} C_VEL
LIN {X 0,Y 488.732,Z 523.61,A -85,B 0,C 180,E1 -6603.483,E2 -6603.483} C_VEL
LIN {X 0,Y 488.683,Z 523.61,A -85,B 0,C 180,E1 -6606.354,E2 -6606.354} C_VEL
LIN {X 0,Y 488.74,Z 523.609,A -85,B 0,C 180,E1 -6609.249,E2 -6609.249} C_VEL
LIN {X 0,Y 488.69,Z 523.609,A -85,B 0,C 180,E1 -6612.524,E2 -6612.524} C_VEL
LIN {X 0,Y 488.706,Z 523.612,A -85,B 0,C 180,E1 -6615.197,E2 -6615.197} C_VEL
LIN {X 0,Y 488.705,Z 523.606,A -85,B 0,C 180,E1 -6618.398,E2 -6618.398} C_VEL
LIN {X 0,Y 488.734,Z 523.604,A -85,B 0,C 180,E1 -6620.941,E2 -6620.941} C_VEL
LIN {X 0,Y 488.679,Z 523.612,A -85,B 0,C 180,E1 -6623.868,E2 -6623.868} C_VEL
LIN {X 0,Y 488.731,Z 523.603,A -85,B 0,C 180,E1 -6626.876,E2 -6626.876} C_VEL
LIN {X 0,Y 488.726,Z 523.607,A -85,B 0,C 180,E1 -6629.78,E2 -6629.78} C_VEL
LIN {X 0,Y 488.79,Z 523.596,A -85,B 0,C 180,E1 -6633.054,E2 -6633.054} C_VEL
LIN {X 0,Y 488.684,Z 523.605,A -85,B 0,C 180,E1 -6636.254,E2 -6636.254} C_VEL
LIN {X 0,Y 488.736,Z 523.607,A -85,B 0,C 180,E1 -6639.175,E2 -6639.175} C_VEL
LIN {X 0,Y 488.749,Z 523.606,A -85,B 0,C 180,E1 -6641.627,E2 -6641.627} C_VEL
LIN {X 0,Y 488.754,Z 523.599,A -85,B 0,C 180,E1 -6644.999,E2 -6644.999} C_VEL
LIN {X 0,Y 488.82,Z 523.588,A -85,B 0,C 180,E1 -6648.387,E2 -6648.387} C_VEL
LIN {X 0,Y 488.808,Z 523.595,A -85,B 0,C 180,E1 -6651.733,E2 -6651.733} C_VEL
LIN {X 0,Y 488.846,Z 523.588,A -85,B 0,C 180,E1 -6654.224,E2 -6654.224} C_VEL
LIN {X 0,Y 488.951,Z 523.581,A -85,B 0,C 180,E1 -6657.528,E2 -6657.528} C_VEL
LIN {X 0,Y 488.958,Z 523.576,A -85,B 0,C 180,E1 -6660,E2 -6660} C_VEL
LIN {X 0,Y 488.951,Z 523.574,A -85,B 0,C 180,E1 -6662.471,E2 -6662.471} C_VEL
LIN {X 0,Y 488.859,Z 523.591,A -85,B 0,C 180,E1 -6665.775,E2 -6665.775} C_VEL
LIN {X 0,Y 488.807,Z 523.594,A -85,B 0,C 180,E1 -6668.266,E2 -6668.266} C_VEL
LIN {X 0,Y 488.821,Z 523.597,A -85,B 0,C 180,E1 -6671.612,E2 -6671.612} C_VEL
LIN {X 0,Y 488.749,Z 523.605,A -85,B 0,C 180,E1 -6675,E2 -6675} C_VEL
LIN {X 0,Y 488.742,Z 523.603,A -85,B 0,C 180,E1 -6678.442,E2 -6678.442} C_VEL
LIN {X 0,Y 488.695,Z 523.612,A -85,B 0,C 180,E1 -6681.071,E2 -6681.071} C_VEL
LIN {X 0,Y 488.681,Z 523.615,A -85,B 0,C 180,E1 -6683.746,E2 -6683.746} C_VEL
LIN {X 0,Y 488.786,Z 523.602,A -85,B 0,C 180,E1 -6686.946,E2 -6686.946} C_VEL
LIN {X 0,Y 488.768,Z 523.662,A -85,B 0,C 180,E1 -6688.547,E2 -6688.547} C_VEL
LIN {X 0,Y 489.95,Z 530.923,A -85,B 0,C 180,E1 -6690.135,E2 -6690.135} C_VEL
LIN {X 0,Y 489.439,Z 545.198,A -85,B 0,C 180,E1 -6693.069,E2 -6693.069} C_VEL
LIN {X 0,Y 489.341,Z 548.725,A -85,B 0,C 180,E1 -6693.789,E2 -6693.789} C_VEL
LIN {X 0,Y 491.782,Z 562.124,A -85,B 0,C 180,E1 -6694.088,E2 -6694.088} C_VEL
LIN {X 0,Y 491.091,Z 655.439,A -85,B 0,C 180,E1 -6695.495,E2 -6695.495} C_VEL
LIN {X 0,Y 490.865,Z 668.165,A -85,B 0,C 180,E1 -6695.842,E2 -6695.842} C_VEL
LIN {X 0,Y 490.56,Z 679.988,A -85,B 0,C 180,E1 -6696.316,E2 -6696.316} C_VEL
LIN {X 0,Y 490.196,Z 691.952,A -85,B 0,C 180,E1 -6696.961,E2 -6696.961} C_VEL
LIN {X 0,Y 489.786,Z 702.861,A -85,B 0,C 180,E1 -6697.723,E2 -6697.723} C_VEL
LIN {X 0,Y 489.398,Z 713.525,A -85,B 0,C 180,E1 -6698.658,E2 -6698.658} C_VEL
LIN {X 0,Y 488.969,Z 723.672,A -85,B 0,C 180,E1 -6699.762,E2 -6699.762} C_VEL
LIN {X 0,Y 488.674,Z 731.891,A -85,B 0,C 180,E1 -6700.871,E2 -6700.871} C_VEL
LIN {X 0,Y 488.338,Z 739.001,A -85,B 0,C 180,E1 -6702.044,E2 -6702.044} C_VEL
LIN {X 0,Y 488.186,Z 745.816,A -85,B 0,C 180,E1 -6703.459,E2 -6703.459} C_VEL
LIN {X 0,Y 488.06,Z 749.8,A -85,B 0,C 180,E1 -6704.505,E2 -6704.505} C_VEL
LIN {X 0,Y 487.292,Z 751.924,A -85,B 0,C 180,E1 -6705.149,E2 -6705.149} C_VEL
LIN {X 0,Y 484.327,Z 754.838,A -85,B 0,C 180,E1 -6706.212,E2 -6706.212} C_VEL
LIN {X 0,Y 481.865,Z 756.648,A -85,B 0,C 180,E1 -6707.085,E2 -6707.085} C_VEL
LIN {X 0,Y 480.799,Z 757.704,A -85,B 0,C 180,E1 -6707.769,E2 -6707.769} C_VEL
LIN {X 0,Y 480.705,Z 757.977,A -85,B 0,C 180,E1 -6708.001,E2 -6708.001} C_VEL
LIN {X 0,Y 480.657,Z 759.087,A -85,B 0,C 180,E1 -6709.492,E2 -6709.492} C_VEL
LIN {X 0,Y 480.683,Z 758.869,A -85,B 0,C 180,E1 -6711.048,E2 -6711.048} C_VEL
LIN {X 0,Y 480.737,Z 757.934,A -85,B 0,C 180,E1 -6712.132,E2 -6712.132} C_VEL
LIN {X 0,Y 480.785,Z 755.742,A -85,B 0,C 180,E1 -6713.511,E2 -6713.511} C_VEL
LIN {X 0,Y 480.89,Z 752.284,A -85,B 0,C 180,E1 -6714.926,E2 -6714.926} C_VEL
LIN {X 0,Y 481.047,Z 747.347,A -85,B 0,C 180,E1 -6716.382,E2 -6716.382} C_VEL
LIN {X 0,Y 481.305,Z 740.631,A -85,B 0,C 180,E1 -6717.877,E2 -6717.877} C_VEL
LIN {X 0,Y 481.549,Z 734.014,A -85,B 0,C 180,E1 -6719.04,E2 -6719.04} C_VEL
LIN {X 0,Y 481.905,Z 725.353,A -85,B 0,C 180,E1 -6720.276,E2 -6720.276} C_VEL
LIN {X 0,Y 482.296,Z 715.824,A -85,B 0,C 180,E1 -6721.378,E2 -6721.378} C_VEL
LIN {X 0,Y 482.704,Z 705.458,A -85,B 0,C 180,E1 -6722.341,E2 -6722.341} C_VEL
LIN {X 0,Y 483.203,Z 693.813,A -85,B 0,C 180,E1 -6723.201,E2 -6723.201} C_VEL
LIN {X 0,Y 483.567,Z 682.382,A -85,B 0,C 180,E1 -6723.862,E2 -6723.862} C_VEL
LIN {X 0,Y 483.943,Z 669.631,A -85,B 0,C 180,E1 -6724.404,E2 -6724.404} C_VEL
LIN {X 0,Y 484.205,Z 656.014,A -85,B 0,C 180,E1 -6724.793,E2 -6724.793} C_VEL
LIN {X 0,Y 484.883,Z 562.29,A -85,B 0,C 180,E1 -6726.232,E2 -6726.232} C_VEL
LIN {X 0,Y 482.327,Z 548.607,A -85,B 0,C 180,E1 -6726.548,E2 -6726.548} C_VEL
LIN {X 0,Y 482.884,Z 533.003,A -85,B 0,C 180,E1 -6729.779,E2 -6729.779} C_VEL
LIN {X 0,Y 482.34,Z 527.984,A -85,B 0,C 180,E1 -6730.864,E2 -6730.864} C_VEL
LIN {X 0,Y 481.742,Z 524.479,A -85,B 0,C 180,E1 -6731.649,E2 -6731.649} C_VEL
LIN {X 0,Y 481.737,Z 524.481,A -85,B 0,C 180,E1 -6734.777,E2 -6734.777} C_VEL
LIN {X 0,Y 481.746,Z 524.473,A -85,B 0,C 180,E1 -6738.216,E2 -6738.216} C_VEL
LIN {X 0,Y 481.759,Z 524.47,A -85,B 0,C 180,E1 -6741.613,E2 -6741.613} C_VEL
LIN {X 0,Y 481.805,Z 524.465,A -85,B 0,C 180,E1 -6744.141,E2 -6744.141} C_VEL
LIN {X 0,Y 481.926,Z 524.45,A -85,B 0,C 180,E1 -6747.494,E2 -6747.494} C_VEL
LIN {X 0,Y 481.903,Z 524.459,A -85,B 0,C 180,E1 -6750.837,E2 -6750.837} C_VEL
LIN {X 0,Y 481.926,Z 524.452,A -85,B 0,C 180,E1 -6752.509,E2 -6752.509} C_VEL
LIN {X 0,Y 481.806,Z 524.464,A -85,B 0,C 180,E1 -6755.862,E2 -6755.862} C_VEL
LIN {X 0,Y 481.761,Z 524.471,A -85,B 0,C 180,E1 -6758.389,E2 -6758.389} C_VEL
LIN {X 0,Y 481.75,Z 524.471,A -85,B 0,C 180,E1 -6761.786,E2 -6761.786} C_VEL
LIN {X 0,Y 481.742,Z 524.479,A -85,B 0,C 180,E1 -6765.225,E2 -6765.225} C_VEL
LIN {X 0,Y 481.708,Z 524.479,A -85,B 0,C 180,E1 -6768.723,E2 -6768.723} C_VEL
LIN {X 0,Y 481.645,Z 524.489,A -85,B 0,C 180,E1 -6771.396,E2 -6771.396} C_VEL
LIN {X 0,Y 481.67,Z 524.481,A -85,B 0,C 180,E1 -6774.115,E2 -6774.115} C_VEL
LIN {X 0,Y 481.747,Z 524.479,A -85,B 0,C 180,E1 -6777.14,E2 -6777.14} C_VEL
LIN {X 0,Y 481.68,Z 524.482,A -85,B 0,C 180,E1 -6779.742,E2 -6779.742} C_VEL
LIN {X 0,Y 481.673,Z 524.482,A -85,B 0,C 180,E1 -6782.675,E2 -6782.675} C_VEL
LIN {X 0,Y 481.638,Z 524.488,A -85,B 0,C 180,E1 -6785.711,E2 -6785.711} C_VEL
LIN {X 0,Y 481.673,Z 524.483,A -85,B 0,C 180,E1 -6788.86,E2 -6788.86} C_VEL
LIN {X 0,Y 481.665,Z 524.483,A -85,B 0,C 180,E1 -6791.915,E2 -6791.915} C_VEL
LIN {X 0,Y 481.663,Z 524.482,A -85,B 0,C 180,E1 -6794.458,E2 -6794.458} C_VEL
LIN {X 0,Y 481.65,Z 524.486,A -85,B 0,C 180,E1 -6797.84,E2 -6797.84} C_VEL
LIN {X 0,Y 481.684,Z 524.479,A -85,B 0,C 180,E1 -6800.652,E2 -6800.652} C_VEL
LIN {X 0,Y 481.631,Z 524.494,A -85,B 0,C 180,E1 -6803.377,E2 -6803.377} C_VEL
LIN {X 0,Y 481.714,Z 524.476,A -85,B 0,C 180,E1 -6806.331,E2 -6806.331} C_VEL
LIN {X 0,Y 481.655,Z 524.49,A -85,B 0,C 180,E1 -6809.418,E2 -6809.418} C_VEL
LIN {X 0,Y 481.704,Z 524.478,A -85,B 0,C 180,E1 -6812.169,E2 -6812.169} C_VEL
LIN {X 0,Y 481.717,Z 524.476,A -85,B 0,C 180,E1 -6814.97,E2 -6814.97} C_VEL
LIN {X 0,Y 481.655,Z 524.49,A -85,B 0,C 180,E1 -6817.706,E2 -6817.706} C_VEL
LIN {X 0,Y 481.71,Z 524.476,A -85,B 0,C 180,E1 -6820.394,E2 -6820.394} C_VEL
LIN {X 0,Y 481.685,Z 524.48,A -85,B 0,C 180,E1 -6823.034,E2 -6823.034} C_VEL
LIN {X 0,Y 481.696,Z 524.486,A -85,B 0,C 180,E1 -6825.639,E2 -6825.639} C_VEL
LIN {X 0,Y 481.757,Z 524.472,A -85,B 0,C 180,E1 -6828.216,E2 -6828.216} C_VEL
LIN {X 0,Y 481.768,Z 524.476,A -85,B 0,C 180,E1 -6831.612,E2 -6831.612} C_VEL
LIN {X 0,Y 481.817,Z 524.466,A -85,B 0,C 180,E1 -6834.14,E2 -6834.14} C_VEL
LIN {X 0,Y 481.934,Z 524.452,A -85,B 0,C 180,E1 -6837.493,E2 -6837.493} C_VEL
LIN {X 0,Y 481.893,Z 524.453,A -85,B 0,C 180,E1 -6840.836,E2 -6840.836} C_VEL
LIN {X 0,Y 481.934,Z 524.449,A -85,B 0,C 180,E1 -6842.508,E2 -6842.508} C_VEL
LIN {X 0,Y 481.823,Z 524.471,A -85,B 0,C 180,E1 -6845.861,E2 -6845.861} C_VEL
LIN {X 0,Y 481.768,Z 524.471,A -85,B 0,C 180,E1 -6848.389,E2 -6848.389} C_VEL
LIN {X 0,Y 481.758,Z 524.476,A -85,B 0,C 180,E1 -6851.785,E2 -6851.785} C_VEL
LIN {X 0,Y 481.75,Z 524.471,A -85,B 0,C 180,E1 -6855.224,E2 -6855.224} C_VEL
LIN {X 0,Y 481.716,Z 524.476,A -85,B 0,C 180,E1 -6858.722,E2 -6858.722} C_VEL
LIN {X 0,Y 481.653,Z 524.484,A -85,B 0,C 180,E1 -6861.395,E2 -6861.395} C_VEL
LIN {X 0,Y 481.669,Z 524.489,A -85,B 0,C 180,E1 -6864.114,E2 -6864.114} C_VEL
LIN {X 0,Y 481.754,Z 524.47,A -85,B 0,C 180,E1 -6867.139,E2 -6867.139} C_VEL
LIN {X 0,Y 481.686,Z 524.482,A -85,B 0,C 180,E1 -6869.741,E2 -6869.741} C_VEL
LIN {X 0,Y 481.678,Z 524.482,A -85,B 0,C 180,E1 -6872.674,E2 -6872.674} C_VEL
LIN {X 0,Y 481.648,Z 524.486,A -85,B 0,C 180,E1 -6875.709,E2 -6875.709} C_VEL
LIN {X 0,Y 481.678,Z 524.481,A -85,B 0,C 180,E1 -6878.859,E2 -6878.859} C_VEL
LIN {X 0,Y 481.653,Z 524.487,A -85,B 0,C 180,E1 -6881.912,E2 -6881.912} C_VEL
LIN {X 0,Y 481.661,Z 524.488,A -85,B 0,C 180,E1 -6884.458,E2 -6884.458} C_VEL
LIN {X 0,Y 481.655,Z 524.485,A -85,B 0,C 180,E1 -6887.839,E2 -6887.839} C_VEL
LIN {X 0,Y 481.687,Z 524.483,A -85,B 0,C 180,E1 -6890.651,E2 -6890.651} C_VEL
LIN {X 0,Y 481.634,Z 524.485,A -85,B 0,C 180,E1 -6893.376,E2 -6893.376} C_VEL
LIN {X 0,Y 481.717,Z 524.483,A -85,B 0,C 180,E1 -6896.329,E2 -6896.329} C_VEL
LIN {X 0,Y 481.657,Z 524.485,A -85,B 0,C 180,E1 -6899.417,E2 -6899.417} C_VEL
LIN {X 0,Y 481.707,Z 524.483,A -85,B 0,C 180,E1 -6902.167,E2 -6902.167} C_VEL
LIN {X 0,Y 481.771,Z 524.657,A -85,B 0,C 180,E1 -6904.649,E2 -6904.649} C_VEL
LIN {X 0,Y 483.709,Z 535.04,A -85,B 0,C 180,E1 -6906.623,E2 -6906.623} C_VEL
LIN {X 0,Y 483.459,Z 545.593,A -85,B 0,C 180,E1 -6908.492,E2 -6908.492} C_VEL
LIN {X 0,Y 482.711,Z 564.381,A -85,B 0,C 180,E1 -6911.757,E2 -6911.757} C_VEL
LIN {X 0,Y 482.355,Z 574.618,A -85,B 0,C 180,E1 -6913.498,E2 -6913.498} C_VEL
LIN {X 0,Y 484.897,Z 590.868,A -85,B 0,C 180,E1 -6913.836,E2 -6913.836} C_VEL
LIN {X 0,Y 484.213,Z 683.501,A -85,B 0,C 180,E1 -6915.258,E2 -6915.258} C_VEL
LIN {X 0,Y 483.82,Z 697.202,A -85,B 0,C 180,E1 -6915.649,E2 -6915.649} C_VEL
LIN {X 0,Y 483.474,Z 709.541,A -85,B 0,C 180,E1 -6916.175,E2 -6916.175} C_VEL
LIN {X 0,Y 483.027,Z 721.395,A -85,B 0,C 180,E1 -6916.859,E2 -6916.859} C_VEL
LIN {X 0,Y 482.634,Z 732.8,A -85,B 0,C 180,E1 -6917.703,E2 -6917.703} C_VEL
LIN {X 0,Y 482.212,Z 743.091,A -85,B 0,C 180,E1 -6918.652,E2 -6918.652} C_VEL
LIN {X 0,Y 481.779,Z 752.329,A -85,B 0,C 180,E1 -6919.705,E2 -6919.705} C_VEL
LIN {X 0,Y 481.428,Z 761.319,A -85,B 0,C 180,E1 -6920.97,E2 -6920.97} C_VEL
LIN {X 0,Y 481.19,Z 768.558,A -85,B 0,C 180,E1 -6922.234,E2 -6922.234} C_VEL
LIN {X 0,Y 480.984,Z 774.406,A -85,B 0,C 180,E1 -6923.515,E2 -6923.515} C_VEL
LIN {X 0,Y 480.903,Z 779.506,A -85,B 0,C 180,E1 -6924.968,E2 -6924.968} C_VEL
LIN {X 0,Y 480.835,Z 781.81,A -85,B 0,C 180,E1 -6925.808,E2 -6925.808} C_VEL
LIN {X 0,Y 480.89,Z 783.683,A -85,B 0,C 180,E1 -6926.648,E2 -6926.648} C_VEL
LIN {X 0,Y 480.823,Z 785.083,A -85,B 0,C 180,E1 -6927.486,E2 -6927.486} C_VEL
LIN {X 0,Y 480.792,Z 786.081,A -85,B 0,C 180,E1 -6928.324,E2 -6928.324} C_VEL
LIN {X 0,Y 480.76,Z 786.688,A -85,B 0,C 180,E1 -6929.161,E2 -6929.161} C_VEL
LIN {X 0,Y 480.743,Z 786.903,A -85,B 0,C 180,E1 -6929.999,E2 -6929.999} C_VEL
LIN {X 0,Y 480.76,Z 786.684,A -85,B 0,C 180,E1 -6930.836,E2 -6930.836} C_VEL
LIN {X 0,Y 480.792,Z 786.071,A -85,B 0,C 180,E1 -6931.674,E2 -6931.674} C_VEL
LIN {X 0,Y 480.823,Z 785.068,A -85,B 0,C 180,E1 -6932.512,E2 -6932.512} C_VEL
LIN {X 0,Y 480.889,Z 783.663,A -85,B 0,C 180,E1 -6933.35,E2 -6933.35} C_VEL
LIN {X 0,Y 480.845,Z 780.705,A -85,B 0,C 180,E1 -6934.61,E2 -6934.61} C_VEL
LIN {X 0,Y 480.958,Z 776.706,A -85,B 0,C 180,E1 -6935.87,E2 -6935.87} C_VEL
LIN {X 0,Y 481.111,Z 770.551,A -85,B 0,C 180,E1 -6937.342,E2 -6937.342} C_VEL
LIN {X 0,Y 481.334,Z 763.827,A -85,B 0,C 180,E1 -6938.606,E2 -6938.606} C_VEL
LIN {X 0,Y 481.641,Z 755.485,A -85,B 0,C 180,E1 -6939.871,E2 -6939.871} C_VEL
LIN {X 0,Y 482.015,Z 746.919,A -85,B 0,C 180,E1 -6940.925,E2 -6940.925} C_VEL
LIN {X 0,Y 482.506,Z 736.34,A -85,B 0,C 180,E1 -6941.978,E2 -6941.978} C_VEL
LIN {X 0,Y 482.841,Z 726.441,A -85,B 0,C 180,E1 -6942.78,E2 -6942.78} C_VEL
LIN {X 0,Y 483.275,Z 714.353,A -85,B 0,C 180,E1 -6943.561,E2 -6943.561} C_VEL
LIN {X 0,Y 483.733,Z 701.139,A -85,B 0,C 180,E1 -6944.191,E2 -6944.191} C_VEL
LIN {X 0,Y 484.092,Z 687.777,A -85,B 0,C 180,E1 -6944.636,E2 -6944.636} C_VEL
LIN {X 0,Y 484.293,Z 672.717,A -85,B 0,C 180,E1 -6944.925,E2 -6944.925} C_VEL
LIN {X 0,Y 484.808,Z 589.902,A -85,B 0,C 180,E1 -6946.179,E2 -6946.179} C_VEL
LIN {X 0,Y 482.343,Z 574.079,A -85,B 0,C 180,E1 -6946.533,E2 -6946.533} C_VEL
LIN {X 0,Y 482.927,Z 556.538,A -85,B 0,C 180,E1 -6949.554,E2 -6949.554} C_VEL
LIN {X 0,Y 483.712,Z 538.858,A -85,B 0,C 180,E1 -6952.644,E2 -6952.644} C_VEL
LIN {X 0,Y 483.686,Z 534.79,A -85,B 0,C 180,E1 -6953.373,E2 -6953.373} C_VEL
LIN {X 0,Y 481.72,Z 524.483,A -85,B 0,C 180,E1 -6955.352,E2 -6955.352} C_VEL
LIN {X 0,Y 481.698,Z 524.487,A -85,B 0,C 180,E1 -6957.83,E2 -6957.83} C_VEL
LIN {X 0,Y 481.644,Z 524.49,A -85,B 0,C 180,E1 -6960.709,E2 -6960.709} C_VEL
LIN {X 0,Y 481.693,Z 524.485,A -85,B 0,C 180,E1 -6963.732,E2 -6963.732} C_VEL
LIN {X 0,Y 481.624,Z 524.49,A -85,B 0,C 180,E1 -6966.745,E2 -6966.745} C_VEL
LIN {X 0,Y 481.684,Z 524.485,A -85,B 0,C 180,E1 -6969.938,E2 -6969.938} C_VEL
LIN {X 0,Y 481.66,Z 524.491,A -85,B 0,C 180,E1 -6973.295,E2 -6973.295} C_VEL
LIN {X 0,Y 481.652,Z 524.492,A -85,B 0,C 180,E1 -6975.639,E2 -6975.639} C_VEL
LIN {X 0,Y 481.661,Z 524.486,A -85,B 0,C 180,E1 -6978.958,E2 -6978.958} C_VEL
LIN {X 0,Y 481.69,Z 524.483,A -85,B 0,C 180,E1 -6981.142,E2 -6981.142} C_VEL
LIN {X 0,Y 481.661,Z 524.484,A -85,B 0,C 180,E1 -6984.793,E2 -6984.793} C_VEL
LIN {X 0,Y 481.665,Z 524.488,A -85,B 0,C 180,E1 -6987.325,E2 -6987.325} C_VEL
LIN {X 0,Y 481.68,Z 524.481,A -85,B 0,C 180,E1 -6990.259,E2 -6990.259} C_VEL
LIN {X 0,Y 481.743,Z 524.475,A -85,B 0,C 180,E1 -6993.111,E2 -6993.111} C_VEL
LIN {X 0,Y 481.668,Z 524.482,A -85,B 0,C 180,E1 -6995.886,E2 -6995.886} C_VEL
LIN {X 0,Y 481.692,Z 524.482,A -85,B 0,C 180,E1 -6999.026,E2 -6999.026} C_VEL
LIN {X 0,Y 481.697,Z 524.479,A -85,B 0,C 180,E1 -7002.158,E2 -7002.158} C_VEL
LIN {X 0,Y 481.733,Z 524.472,A -85,B 0,C 180,E1 -7004.775,E2 -7004.775} C_VEL
LIN {X 0,Y 481.784,Z 524.465,A -85,B 0,C 180,E1 -7008.216,E2 -7008.216} C_VEL
LIN {X 0,Y 481.753,Z 524.475,A -85,B 0,C 180,E1 -7011.611,E2 -7011.611} C_VEL
LIN {X 0,Y 481.807,Z 524.465,A -85,B 0,C 180,E1 -7014.139,E2 -7014.139} C_VEL
LIN {X 0,Y 481.918,Z 524.457,A -85,B 0,C 180,E1 -7017.492,E2 -7017.492} C_VEL
LIN {X 0,Y 481.929,Z 524.452,A -85,B 0,C 180,E1 -7020,E2 -7020} C_VEL
LIN {X 0,Y 481.918,Z 524.45,A -85,B 0,C 180,E1 -7022.507,E2 -7022.507} C_VEL
LIN {X 0,Y 481.817,Z 524.467,A -85,B 0,C 180,E1 -7025.86,E2 -7025.86} C_VEL
LIN {X 0,Y 481.752,Z 524.472,A -85,B 0,C 180,E1 -7028.388,E2 -7028.388} C_VEL
LIN {X 0,Y 481.783,Z 524.472,A -85,B 0,C 180,E1 -7031.784,E2 -7031.784} C_VEL
LIN {X 0,Y 481.73,Z 524.483,A -85,B 0,C 180,E1 -7035.224,E2 -7035.224} C_VEL
LIN {X 0,Y 481.7,Z 524.481,A -85,B 0,C 180,E1 -7038.722,E2 -7038.722} C_VEL
LIN {X 0,Y 481.635,Z 524.492,A -85,B 0,C 180,E1 -7041.395,E2 -7041.395} C_VEL
LIN {X 0,Y 481.665,Z 524.486,A -85,B 0,C 180,E1 -7044.113,E2 -7044.113} C_VEL
LIN {X 0,Y 481.74,Z 524.48,A -85,B 0,C 180,E1 -7047.141,E2 -7047.141} C_VEL
LIN {X 0,Y 481.731,Z 524.562,A -85,B 0,C 180,E1 -7048.362,E2 -7048.362} C_VEL
LIN {X 0,Y 483.013,Z 532.528,A -85,B 0,C 180,E1 -7050.131,E2 -7050.131} C_VEL
LIN {X 0,Y 482.442,Z 546.839,A -85,B 0,C 180,E1 -7053.112,E2 -7053.112} C_VEL
LIN {X 0,Y 482.361,Z 548.987,A -85,B 0,C 180,E1 -7053.555,E2 -7053.555} C_VEL
LIN {X 0,Y 484.999,Z 563.572,A -85,B 0,C 180,E1 -7053.877,E2 -7053.877} C_VEL
LIN {X 0,Y 484.23,Z 656.09,A -85,B 0,C 180,E1 -7055.297,E2 -7055.297} C_VEL
LIN {X 0,Y 483.996,Z 668.8,A -85,B 0,C 180,E1 -7055.655,E2 -7055.655} C_VEL
LIN {X 0,Y 483.605,Z 681.601,A -85,B 0,C 180,E1 -7056.185,E2 -7056.185} C_VEL
LIN {X 0,Y 483.225,Z 693.79,A -85,B 0,C 180,E1 -7056.88,E2 -7056.88} C_VEL
LIN {X 0,Y 482.757,Z 704.861,A -85,B 0,C 180,E1 -7057.693,E2 -7057.693} C_VEL
LIN {X 0,Y 482.393,Z 714.939,A -85,B 0,C 180,E1 -7058.615,E2 -7058.615} C_VEL
LIN {X 0,Y 481.96,Z 724.034,A -85,B 0,C 180,E1 -7059.633,E2 -7059.633} C_VEL
LIN {X 0,Y 481.627,Z 732.589,A -85,B 0,C 180,E1 -7060.816,E2 -7060.816} C_VEL
LIN {X 0,Y 481.259,Z 740.641,A -85,B 0,C 180,E1 -7062.202,E2 -7062.202} C_VEL
LIN {X 0,Y 481.138,Z 745.978,A -85,B 0,C 180,E1 -7063.355,E2 -7063.355} C_VEL
LIN {X 0,Y 480.979,Z 750.38,A -85,B 0,C 180,E1 -7064.536,E2 -7064.536} C_VEL
LIN {X 0,Y 480.843,Z 753.874,A -85,B 0,C 180,E1 -7065.74,E2 -7065.74} C_VEL
LIN {X 0,Y 480.781,Z 756.477,A -85,B 0,C 180,E1 -7066.961,E2 -7066.961} C_VEL
LIN {X 0,Y 480.705,Z 757.977,A -85,B 0,C 180,E1 -7068.001,E2 -7068.001} C_VEL
LIN {X 0,Y 480.007,Z 758.697,A -85,B 0,C 180,E1 -7068.697,E2 -7068.697} C_VEL
LIN {X 0,Y 477.108,Z 759.287,A -85,B 0,C 180,E1 -7069.831,E2 -7069.831} C_VEL
LIN {X 0,Y 474.687,Z 759.218,A -85,B 0,C 180,E1 -7070.747,E2 -7070.747} C_VEL
LIN {X 0,Y 473.672,Z 758.831,A -85,B 0,C 180,E1 -7071.453,E2 -7071.453} C_VEL
LIN {X 0,Y 473.602,Z 758.609,A -85,B 0,C 180,E1 -7071.691,E2 -7071.691} C_VEL
LIN {X 0,Y 473.69,Z 756.529,A -85,B 0,C 180,E1 -7073.242,E2 -7073.242} C_VEL
LIN {X 0,Y 473.804,Z 753.395,A -85,B 0,C 180,E1 -7074.668,E2 -7074.668} C_VEL
LIN {X 0,Y 473.925,Z 748.794,A -85,B 0,C 180,E1 -7076.143,E2 -7076.143} C_VEL
LIN {X 0,Y 474.177,Z 742.473,A -85,B 0,C 180,E1 -7077.652,E2 -7077.652} C_VEL
LIN {X 0,Y 474.475,Z 735.138,A -85,B 0,C 180,E1 -7079.022,E2 -7079.022} C_VEL
LIN {X 0,Y 474.848,Z 726.653,A -85,B 0,C 180,E1 -7080.278,E2 -7080.278} C_VEL
LIN {X 0,Y 475.283,Z 717.312,A -85,B 0,C 180,E1 -7081.399,E2 -7081.399} C_VEL
LIN {X 0,Y 475.707,Z 706.742,A -85,B 0,C 180,E1 -7082.427,E2 -7082.427} C_VEL
LIN {X 0,Y 476.198,Z 696.08,A -85,B 0,C 180,E1 -7083.249,E2 -7083.249} C_VEL
LIN {X 0,Y 476.639,Z 683.556,A -85,B 0,C 180,E1 -7084.007,E2 -7084.007} C_VEL
LIN {X 0,Y 477.031,Z 671.125,A -85,B 0,C 180,E1 -7084.563,E2 -7084.563} C_VEL
LIN {X 0,Y 477.301,Z 657.588,A -85,B 0,C 180,E1 -7084.971,E2 -7084.971} C_VEL
LIN {X 0,Y 477.538,Z 633.294,A -85,B 0,C 180,E1 -7085.376,E2 -7085.376} C_VEL
LIN {X 0,Y 477.994,Z 562.591,A -85,B 0,C 180,E1 -7086.468,E2 -7086.468} C_VEL
LIN {X 0,Y 475.398,Z 548.796,A -85,B 0,C 180,E1 -7086.794,E2 -7086.794} C_VEL
LIN {X 0,Y 475.942,Z 533.89,A -85,B 0,C 180,E1 -7089.922,E2 -7089.922} C_VEL
LIN {X 0,Y 474.719,Z 525.408,A -85,B 0,C 180,E1 -7091.799,E2 -7091.799} C_VEL
LIN {X 0,Y 474.694,Z 525.358,A -85,B 0,C 180,E1 -7094.546,E2 -7094.546} C_VEL
LIN {X 0,Y 474.699,Z 525.35,A -85,B 0,C 180,E1 -7098.039,E2 -7098.039} C_VEL
LIN {X 0,Y 474.724,Z 525.347,A -85,B 0,C 180,E1 -7101.488,E2 -7101.488} C_VEL
LIN {X 0,Y 474.767,Z 525.341,A -85,B 0,C 180,E1 -7104.054,E2 -7104.054} C_VEL
LIN {X 0,Y 474.892,Z 525.327,A -85,B 0,C 180,E1 -7107.457,E2 -7107.457} C_VEL
LIN {X 0,Y 474.909,Z 525.323,A -85,B 0,C 180,E1 -7110.001,E2 -7110.001} C_VEL
LIN {X 0,Y 474.892,Z 525.328,A -85,B 0,C 180,E1 -7112.546,E2 -7112.546} C_VEL
LIN {X 0,Y 474.768,Z 525.341,A -85,B 0,C 180,E1 -7115.949,E2 -7115.949} C_VEL
LIN {X 0,Y 474.726,Z 525.348,A -85,B 0,C 180,E1 -7118.515,E2 -7118.515} C_VEL
LIN {X 0,Y 474.703,Z 525.349,A -85,B 0,C 180,E1 -7121.964,E2 -7121.964} C_VEL
LIN {X 0,Y 474.699,Z 525.353,A -85,B 0,C 180,E1 -7125.457,E2 -7125.457} C_VEL
LIN {X 0,Y 474.662,Z 525.361,A -85,B 0,C 180,E1 -7129.011,E2 -7129.011} C_VEL
LIN {X 0,Y 474.588,Z 525.365,A -85,B 0,C 180,E1 -7131.73,E2 -7131.73} C_VEL
LIN {X 0,Y 474.654,Z 525.356,A -85,B 0,C 180,E1 -7134.494,E2 -7134.494} C_VEL
LIN {X 0,Y 474.682,Z 525.358,A -85,B 0,C 180,E1 -7137.335,E2 -7137.335} C_VEL
LIN {X 0,Y 474.606,Z 525.361,A -85,B 0,C 180,E1 -7140.231,E2 -7140.231} C_VEL
LIN {X 0,Y 474.644,Z 525.365,A -85,B 0,C 180,E1 -7143.221,E2 -7143.221} C_VEL
LIN {X 0,Y 474.59,Z 525.363,A -85,B 0,C 180,E1 -7146.325,E2 -7146.325} C_VEL
LIN {X 0,Y 474.63,Z 525.362,A -85,B 0,C 180,E1 -7149.649,E2 -7149.649} C_VEL
LIN {X 0,Y 474.638,Z 525.36,A -85,B 0,C 180,E1 -7152.933,E2 -7152.933} C_VEL
LIN {X 0,Y 474.612,Z 525.362,A -85,B 0,C 180,E1 -7155.896,E2 -7155.896} C_VEL
LIN {X 0,Y 474.63,Z 525.361,A -85,B 0,C 180,E1 -7159.042,E2 -7159.042} C_VEL
LIN {X 0,Y 474.613,Z 525.365,A -85,B 0,C 180,E1 -7161.705,E2 -7161.705} C_VEL
LIN {X 0,Y 474.628,Z 525.359,A -85,B 0,C 180,E1 -7164.727,E2 -7164.727} C_VEL
LIN {X 0,Y 474.64,Z 525.361,A -85,B 0,C 180,E1 -7167.789,E2 -7167.789} C_VEL
LIN {X 0,Y 474.628,Z 525.359,A -85,B 0,C 180,E1 -7170.886,E2 -7170.886} C_VEL
LIN {X 0,Y 474.664,Z 525.362,A -85,B 0,C 180,E1 -7173.629,E2 -7173.629} C_VEL
LIN {X 0,Y 474.641,Z 525.356,A -85,B 0,C 180,E1 -7176.642,E2 -7176.642} C_VEL
LIN {X 0,Y 474.659,Z 525.357,A -85,B 0,C 180,E1 -7180.09,E2 -7180.09} C_VEL
LIN {X 0,Y 474.645,Z 525.356,A -85,B 0,C 180,E1 -7182.775,E2 -7182.775} C_VEL
LIN {X 0,Y 474.654,Z 525.36,A -85,B 0,C 180,E1 -7185.422,E2 -7185.422} C_VEL
LIN {X 0,Y 474.71,Z 525.352,A -85,B 0,C 180,E1 -7188.038,E2 -7188.038} C_VEL
LIN {X 0,Y 474.733,Z 525.35,A -85,B 0,C 180,E1 -7191.487,E2 -7191.487} C_VEL
LIN {X 0,Y 474.779,Z 525.344,A -85,B 0,C 180,E1 -7194.053,E2 -7194.053} C_VEL
LIN {X 0,Y 474.9,Z 525.328,A -85,B 0,C 180,E1 -7197.456,E2 -7197.456} C_VEL
LIN {X 0,Y 474.918,Z 525.328,A -85,B 0,C 180,E1 -7200,E2 -7200} C_VEL
LIN {X 0,Y 474.9,Z 525.325,A -85,B 0,C 180,E1 -7202.545,E2 -7202.545} C_VEL
LIN {X 0,Y 474.786,Z 525.346,A -85,B 0,C 180,E1 -7205.948,E2 -7205.948} C_VEL
LIN {X 0,Y 474.734,Z 525.346,A -85,B 0,C 180,E1 -7208.514,E2 -7208.514} C_VEL
LIN {X 0,Y 474.712,Z 525.356,A -85,B 0,C 180,E1 -7211.963,E2 -7211.963} C_VEL
LIN {X 0,Y 474.707,Z 525.35,A -85,B 0,C 180,E1 -7215.456,E2 -7215.456} C_VEL
LIN {X 0,Y 474.67,Z 525.353,A -85,B 0,C 180,E1 -7219.01,E2 -7219.01} C_VEL
LIN {X 0,Y 474.596,Z 525.366,A -85,B 0,C 180,E1 -7221.729,E2 -7221.729} C_VEL
LIN {X 0,Y 474.648,Z 525.359,A -85,B 0,C 180,E1 -7224.494,E2 -7224.494} C_VEL
LIN {X 0,Y 474.689,Z 525.351,A -85,B 0,C 180,E1 -7227.334,E2 -7227.334} C_VEL
LIN {X 0,Y 474.612,Z 525.361,A -85,B 0,C 180,E1 -7230.81,E2 -7230.81} C_VEL
LIN {X 0,Y 474.645,Z 525.362,A -85,B 0,C 180,E1 -7233.984,E2 -7233.984} C_VEL
LIN {X 0,Y 474.581,Z 525.365,A -85,B 0,C 180,E1 -7236.899,E2 -7236.899} C_VEL
LIN {X 0,Y 474.62,Z 525.361,A -85,B 0,C 180,E1 -7239.645,E2 -7239.645} C_VEL
LIN {X 0,Y 474.607,Z 525.369,A -85,B 0,C 180,E1 -7242.233,E2 -7242.233} C_VEL
LIN {X 0,Y 474.624,Z 525.359,A -85,B 0,C 180,E1 -7245.297,E2 -7245.297} C_VEL
LIN {X 0,Y 474.628,Z 525.365,A -85,B 0,C 180,E1 -7248.214,E2 -7248.214} C_VEL
LIN {X 0,Y 474.651,Z 525.362,A -85,B 0,C 180,E1 -7250.454,E2 -7250.454} C_VEL
LIN {X 0,Y 474.596,Z 525.363,A -85,B 0,C 180,E1 -7253.676,E2 -7253.676} C_VEL
LIN {X 0,Y 474.65,Z 525.359,A -85,B 0,C 180,E1 -7256.779,E2 -7256.779} C_VEL
LIN {X 0,Y 474.612,Z 525.363,A -85,B 0,C 180,E1 -7259.769,E2 -7259.769} C_VEL
LIN {X 0,Y 474.704,Z 525.356,A -85,B 0,C 180,E1 -7262.679,E2 -7262.679} C_VEL
LIN {X 0,Y 474.696,Z 525.391,A -85,B 0,C 180,E1 -7264.414,E2 -7264.414} C_VEL
LIN {X 0,Y 476.768,Z 536.415,A -85,B 0,C 180,E1 -7266.545,E2 -7266.545} C_VEL
LIN {X 0,Y 476.522,Z 546.52,A -85,B 0,C 180,E1 -7268.363,E2 -7268.363} C_VEL
LIN {X 0,Y 475.723,Z 565.453,A -85,B 0,C 180,E1 -7271.703,E2 -7271.703} C_VEL
LIN {X 0,Y 475.394,Z 574.572,A -85,B 0,C 180,E1 -7273.253,E2 -7273.253} C_VEL
LIN {X 0,Y 478.086,Z 591.619,A -85,B 0,C 180,E1 -7273.615,E2 -7273.615} C_VEL
LIN {X 0,Y 477.36,Z 683.053,A -85,B 0,C 180,E1 -7275.041,E2 -7275.041} C_VEL
LIN {X 0,Y 476.978,Z 696.075,A -85,B 0,C 180,E1 -7275.411,E2 -7275.411} C_VEL
LIN {X 0,Y 476.581,Z 708.126,A -85,B 0,C 180,E1 -7275.916,E2 -7275.916} C_VEL
LIN {X 0,Y 476.132,Z 719.84,A -85,B 0,C 180,E1 -7276.578,E2 -7276.578} C_VEL
LIN {X 0,Y 475.706,Z 730.341,A -85,B 0,C 180,E1 -7277.337,E2 -7277.337} C_VEL
LIN {X 0,Y 475.301,Z 740.706,A -85,B 0,C 180,E1 -7278.268,E2 -7278.268} C_VEL
LIN {X 0,Y 474.83,Z 750.394,A -85,B 0,C 180,E1 -7279.337,E2 -7279.337} C_VEL
LIN {X 0,Y 474.487,Z 758.334,A -85,B 0,C 180,E1 -7280.407,E2 -7280.407} C_VEL
LIN {X 0,Y 474.184,Z 766.092,A -85,B 0,C 180,E1 -7281.69,E2 -7281.69} C_VEL
LIN {X 0,Y 473.938,Z 773.226,A -85,B 0,C 180,E1 -7283.186,E2 -7283.186} C_VEL
LIN {X 0,Y 473.867,Z 777.977,A -85,B 0,C 180,E1 -7284.467,E2 -7284.467} C_VEL
LIN {X 0,Y 473.741,Z 781.603,A -85,B 0,C 180,E1 -7285.745,E2 -7285.745} C_VEL
LIN {X 0,Y 473.797,Z 783.477,A -85,B 0,C 180,E1 -7286.597,E2 -7286.597} C_VEL
LIN {X 0,Y 473.742,Z 784.879,A -85,B 0,C 180,E1 -7287.448,E2 -7287.448} C_VEL
LIN {X 0,Y 473.688,Z 786.485,A -85,B 0,C 180,E1 -7289.149,E2 -7289.149} C_VEL
LIN {X 0,Y 473.669,Z 786.699,A -85,B 0,C 180,E1 -7289.999,E2 -7289.999} C_VEL
LIN {X 0,Y 473.688,Z 786.479,A -85,B 0,C 180,E1 -7290.849,E2 -7290.849} C_VEL
LIN {X 0,Y 473.741,Z 784.86,A -85,B 0,C 180,E1 -7292.55,E2 -7292.55} C_VEL
LIN {X 0,Y 473.797,Z 783.452,A -85,B 0,C 180,E1 -7293.4,E2 -7293.4} C_VEL
LIN {X 0,Y 473.768,Z 780.49,A -85,B 0,C 180,E1 -7294.679,E2 -7294.679} C_VEL
LIN {X 0,Y 473.863,Z 776.485,A -85,B 0,C 180,E1 -7295.958,E2 -7295.958} C_VEL
LIN {X 0,Y 474.023,Z 770.322,A -85,B 0,C 180,E1 -7297.453,E2 -7297.453} C_VEL
LIN {X 0,Y 474.296,Z 763.594,A -85,B 0,C 180,E1 -7298.735,E2 -7298.735} C_VEL
LIN {X 0,Y 474.607,Z 755.247,A -85,B 0,C 180,E1 -7300.019,E2 -7300.019} C_VEL
LIN {X 0,Y 475.02,Z 746.674,A -85,B 0,C 180,E1 -7301.088,E2 -7301.088} C_VEL
LIN {X 0,Y 475.52,Z 736.238,A -85,B 0,C 180,E1 -7302.143,E2 -7302.143} C_VEL
LIN {X 0,Y 475.933,Z 725.896,A -85,B 0,C 180,E1 -7302.991,E2 -7302.991} C_VEL
LIN {X 0,Y 476.354,Z 714.082,A -85,B 0,C 180,E1 -7303.761,E2 -7303.761} C_VEL
LIN {X 0,Y 476.802,Z 702.15,A -85,B 0,C 180,E1 -7304.347,E2 -7304.347} C_VEL
LIN {X 0,Y 477.164,Z 689.292,A -85,B 0,C 180,E1 -7304.799,E2 -7304.799} C_VEL
LIN {X 0,Y 477.426,Z 675.865,A -85,B 0,C 180,E1 -7305.091,E2 -7305.091} C_VEL
LIN {X 0,Y 477.975,Z 590.614,A -85,B 0,C 180,E1 -7306.402,E2 -7306.402} C_VEL
LIN {X 0,Y 475.369,Z 574.006,A -85,B 0,C 180,E1 -7306.76,E2 -7306.76} C_VEL
LIN {X 0,Y 475.95,Z 557.744,A -85,B 0,C 180,E1 -7309.605,E2 -7309.605} C_VEL
LIN {X 0,Y 476.781,Z 539.966,A -85,B 0,C 180,E1 -7312.763,E2 -7312.763} C_VEL
LIN {X 0,Y 476.744,Z 536.178,A -85,B 0,C 180,E1 -7313.453,E2 -7313.453} C_VEL
LIN {X 0,Y 474.665,Z 525.361,A -85,B 0,C 180,E1 -7315.559,E2 -7315.559} C_VEL
LIN {X 0,Y 474.644,Z 525.363,A -85,B 0,C 180,E1 -7318.281,E2 -7318.281} C_VEL
LIN {X 0,Y 474.597,Z 525.37,A -85,B 0,C 180,E1 -7321.216,E2 -7321.216} C_VEL
LIN {X 0,Y 474.629,Z 525.36,A -85,B 0,C 180,E1 -7324.239,E2 -7324.239} C_VEL
LIN {X 0,Y 474.59,Z 525.372,A -85,B 0,C 180,E1 -7327.382,E2 -7327.382} C_VEL
LIN {X 0,Y 474.647,Z 525.365,A -85,B 0,C 180,E1 -7329.65,E2 -7329.65} C_VEL
LIN {X 0,Y 474.63,Z 525.363,A -85,B 0,C 180,E1 -7332.93,E2 -7332.93} C_VEL
LIN {X 0,Y 474.603,Z 525.367,A -85,B 0,C 180,E1 -7335.894,E2 -7335.894} C_VEL
LIN {X 0,Y 474.634,Z 525.363,A -85,B 0,C 180,E1 -7339.038,E2 -7339.038} C_VEL
LIN {X 0,Y 474.609,Z 525.365,A -85,B 0,C 180,E1 -7341.702,E2 -7341.702} C_VEL
LIN {X 0,Y 474.623,Z 525.361,A -85,B 0,C 180,E1 -7344.725,E2 -7344.725} C_VEL
LIN {X 0,Y 474.629,Z 525.362,A -85,B 0,C 180,E1 -7347.787,E2 -7347.787} C_VEL
LIN {X 0,Y 474.623,Z 525.361,A -85,B 0,C 180,E1 -7350.882,E2 -7350.882} C_VEL
LIN {X 0,Y 474.658,Z 525.362,A -85,B 0,C 180,E1 -7353.628,E2 -7353.628} C_VEL
LIN {X 0,Y 474.625,Z 525.356,A -85,B 0,C 180,E1 -7356.64,E2 -7356.64} C_VEL
LIN {X 0,Y 474.647,Z 525.354,A -85,B 0,C 180,E1 -7360.089,E2 -7360.089} C_VEL
LIN {X 0,Y 474.641,Z 525.359,A -85,B 0,C 180,E1 -7362.774,E2 -7362.774} C_VEL
LIN {X 0,Y 474.642,Z 525.363,A -85,B 0,C 180,E1 -7365.42,E2 -7365.42} C_VEL
LIN {X 0,Y 474.728,Z 525.345,A -85,B 0,C 180,E1 -7368.038,E2 -7368.038} C_VEL
LIN {X 0,Y 474.718,Z 525.351,A -85,B 0,C 180,E1 -7371.486,E2 -7371.486} C_VEL
LIN {X 0,Y 474.769,Z 525.342,A -85,B 0,C 180,E1 -7374.052,E2 -7374.052} C_VEL
LIN {X 0,Y 474.885,Z 525.334,A -85,B 0,C 180,E1 -7377.455,E2 -7377.455} C_VEL
LIN {X 0,Y 474.866,Z 525.332,A -85,B 0,C 180,E1 -7380.848,E2 -7380.848} C_VEL
LIN {X 0,Y 474.885,Z 525.327,A -85,B 0,C 180,E1 -7382.544,E2 -7382.544} C_VEL
LIN {X 0,Y 474.778,Z 525.343,A -85,B 0,C 180,E1 -7385.947,E2 -7385.947} C_VEL
LIN {X 0,Y 474.717,Z 525.349,A -85,B 0,C 180,E1 -7388.513,E2 -7388.513} C_VEL
LIN {X 0,Y 474.726,Z 525.35,A -85,B 0,C 180,E1 -7391.961,E2 -7391.961} C_VEL
LIN {X 0,Y 474.668,Z 525.361,A -85,B 0,C 180,E1 -7395.768,E2 -7395.768} C_VEL
LIN {X 0,Y 474.653,Z 525.362,A -85,B 0,C 180,E1 -7399.01,E2 -7399.01} C_VEL
LIN {X 0,Y 474.578,Z 525.371,A -85,B 0,C 180,E1 -7401.729,E2 -7401.729} C_VEL
LIN {X 0,Y 474.647,Z 525.36,A -85,B 0,C 180,E1 -7404.493,E2 -7404.493} C_VEL
LIN {X 0,Y 474.655,Z 525.363,A -85,B 0,C 180,E1 -7407.8,E2 -7407.8} C_VEL
LIN {X 0,Y 474.666,Z 525.419,A -85,B 0,C 180,E1 -7408.16,E2 -7408.16} C_VEL
LIN {X 0,Y 476.041,Z 533.022,A -85,B 0,C 180,E1 -7409.885,E2 -7409.885} C_VEL
LIN {X 0,Y 475.541,Z 545.889,A -85,B 0,C 180,E1 -7412.609,E2 -7412.609} C_VEL
LIN {X 0,Y 475.408,Z 549.112,A -85,B 0,C 180,E1 -7413.286,E2 -7413.286} C_VEL
LIN {X 0,Y 478.169,Z 563.589,A -85,B 0,C 180,E1 -7413.636,E2 -7413.636} C_VEL
LIN {X 0,Y 477.358,Z 656.604,A -85,B 0,C 180,E1 -7415.09,E2 -7415.09} C_VEL
LIN {X 0,Y 477.104,Z 669.625,A -85,B 0,C 180,E1 -7415.467,E2 -7415.467} C_VEL
LIN {X 0,Y 476.721,Z 682.052,A -85,B 0,C 180,E1 -7415.995,E2 -7415.995} C_VEL
LIN {X 0,Y 476.322,Z 694.09,A -85,B 0,C 180,E1 -7416.695,E2 -7416.695} C_VEL
LIN {X 0,Y 475.8,Z 705.382,A -85,B 0,C 180,E1 -7417.538,E2 -7417.538} C_VEL
LIN {X 0,Y 475.414,Z 715.677,A -85,B 0,C 180,E1 -7418.501,E2 -7418.501} C_VEL
LIN {X 0,Y 474.946,Z 724.517,A -85,B 0,C 180,E1 -7419.515,E2 -7419.515} C_VEL
LIN {X 0,Y 474.608,Z 732.654,A -85,B 0,C 180,E1 -7420.658,E2 -7420.658} C_VEL
LIN {X 0,Y 474.264,Z 739.476,A -85,B 0,C 180,E1 -7421.823,E2 -7421.823} C_VEL
LIN {X 0,Y 474.088,Z 745.069,A -85,B 0,C 180,E1 -7422.993,E2 -7422.993} C_VEL
LIN {X 0,Y 473.941,Z 749.677,A -85,B 0,C 180,E1 -7424.183,E2 -7424.183} C_VEL
LIN {X 0,Y 473.746,Z 754.375,A -85,B 0,C 180,E1 -7425.796,E2 -7425.796} C_VEL
LIN {X 0,Y 473.686,Z 756.761,A -85,B 0,C 180,E1 -7426.963,E2 -7426.963} C_VEL
LIN {X 0,Y 473.605,Z 758.357,A -85,B 0,C 180,E1 -7428.107,E2 -7428.107} C_VEL
LIN {X 0,Y 473.569,Z 759.199,A -85,B 0,C 180,E1 -7429.235,E2 -7429.235} C_VEL
LIN {X 0,Y 473.579,Z 759.304,A -85,B 0,C 180,E1 -7430.505,E2 -7430.505} C_VEL
LIN {X 0,Y 473.602,Z 758.609,A -85,B 0,C 180,E1 -7431.691,E2 -7431.691} C_VEL
LIN {X 0,Y 472.976,Z 757.866,A -85,B 0,C 180,E1 -7432.396,E2 -7432.396} C_VEL
LIN {X 0,Y 470.174,Z 756.149,A -85,B 0,C 180,E1 -7433.534,E2 -7433.534} C_VEL
LIN {X 0,Y 467.81,Z 754.27,A -85,B 0,C 180,E1 -7434.438,E2 -7434.438} C_VEL
LIN {X 0,Y 466.827,Z 752.52,A -85,B 0,C 180,E1 -7435.124,E2 -7435.124} C_VEL
LIN {X 0,Y 466.765,Z 751.849,A -85,B 0,C 180,E1 -7435.354,E2 -7435.354} C_VEL
LIN {X 0,Y 466.939,Z 747.328,A -85,B 0,C 180,E1 -7436.678,E2 -7436.678} C_VEL
LIN {X 0,Y 467.183,Z 741.405,A -85,B 0,C 180,E1 -7438.031,E2 -7438.031} C_VEL
LIN {X 0,Y 467.469,Z 734.669,A -85,B 0,C 180,E1 -7439.261,E2 -7439.261} C_VEL
LIN {X 0,Y 467.893,Z 725.579,A -85,B 0,C 180,E1 -7440.596,E2 -7440.596} C_VEL
LIN {X 0,Y 468.335,Z 716.553,A -85,B 0,C 180,E1 -7441.67,E2 -7441.67} C_VEL
LIN {X 0,Y 468.844,Z 706.107,A -85,B 0,C 180,E1 -7442.674,E2 -7442.674} C_VEL
LIN {X 0,Y 469.39,Z 694.441,A -85,B 0,C 180,E1 -7443.565,E2 -7443.565} C_VEL
LIN {X 0,Y 469.824,Z 682.164,A -85,B 0,C 180,E1 -7444.292,E2 -7444.292} C_VEL
LIN {X 0,Y 470.22,Z 669.182,A -85,B 0,C 180,E1 -7444.849,E2 -7444.849} C_VEL
LIN {X 0,Y 470.508,Z 655.772,A -85,B 0,C 180,E1 -7445.234,E2 -7445.234} C_VEL
LIN {X 0,Y 471.261,Z 563.96,A -85,B 0,C 180,E1 -7446.686,E2 -7446.686} C_VEL
LIN {X 0,Y 468.428,Z 548.998,A -85,B 0,C 180,E1 -7447.042,E2 -7447.042} C_VEL
LIN {X 0,Y 468.98,Z 534.77,A -85,B 0,C 180,E1 -7450.068,E2 -7450.068} C_VEL
LIN {X 0,Y 467.629,Z 526.236,A -85,B 0,C 180,E1 -7452,E2 -7452} C_VEL
LIN {X 0,Y 467.602,Z 526.239,A -85,B 0,C 180,E1 -7455.198,E2 -7455.198} C_VEL
LIN {X 0,Y 467.651,Z 526.227,A -85,B 0,C 180,E1 -7457.856,E2 -7457.856} C_VEL
LIN {X 0,Y 467.677,Z 526.226,A -85,B 0,C 180,E1 -7461.358,E2 -7461.358} C_VEL
LIN {X 0,Y 467.732,Z 526.217,A -85,B 0,C 180,E1 -7463.964,E2 -7463.964} C_VEL
LIN {X 0,Y 467.858,Z 526.203,A -85,B 0,C 180,E1 -7467.418,E2 -7467.418} C_VEL
LIN {X 0,Y 467.88,Z 526.199,A -85,B 0,C 180,E1 -7470.001,E2 -7470.001} C_VEL
LIN {X 0,Y 467.858,Z 526.205,A -85,B 0,C 180,E1 -7472.584,E2 -7472.584} C_VEL
LIN {X 0,Y 467.733,Z 526.217,A -85,B 0,C 180,E1 -7476.039,E2 -7476.039} C_VEL
LIN {X 0,Y 467.68,Z 526.227,A -85,B 0,C 180,E1 -7478.644,E2 -7478.644} C_VEL
LIN {X 0,Y 467.655,Z 526.227,A -85,B 0,C 180,E1 -7482.147,E2 -7482.147} C_VEL
LIN {X 0,Y 467.638,Z 526.23,A -85,B 0,C 180,E1 -7485.696,E2 -7485.696} C_VEL
LIN {X 0,Y 467.613,Z 526.236,A -85,B 0,C 180,E1 -7488.764,E2 -7488.764} C_VEL
LIN {X 0,Y 467.58,Z 526.243,A -85,B 0,C 180,E1 -7491.269,E2 -7491.269} C_VEL
LIN {X 0,Y 467.57,Z 526.238,A -85,B 0,C 180,E1 -7493.945,E2 -7493.945} C_VEL
LIN {X 0,Y 467.617,Z 526.235,A -85,B 0,C 180,E1 -7496.801,E2 -7496.801} C_VEL
LIN {X 0,Y 467.555,Z 526.241,A -85,B 0,C 180,E1 -7499.739,E2 -7499.739} C_VEL
